LIN {X 0,Y 561.925,Z 555.197,A -85,B 0,C 180,E1 23264.855,E2 23264.855} C_VEL
LIN {X 0,Y 556.001,Z 546.029,A -85,B 0,C 180,E1 23264.105,E2 23264.105} C_VEL
LIN {X 0,Y 547.752,Z 527.565,A -85,B 0,C 180,E1 23261.432,E2 23261.432} C_VEL
LIN {X 0,Y 541.209,Z 514.277,A -85,B 0,C 180,E1 23259.278,E2 23259.278} C_VEL
LIN {X 0,Y 538.784,Z 509.459,A -85,B 0,C 180,E1 23258.452,E2 23258.452} C_VEL
LIN {X 0,Y 537.627,Z 506.4,A -85,B 0,C 180,E1 23257.909,E2 23257.909} C_VEL
LIN {X 0,Y 537.605,Z 506.203,A -85,B 0,C 180,E1 23254.522,E2 23254.522} C_VEL
LIN {X 0,Y 537.577,Z 506.243,A -85,B 0,C 180,E1 23251.137,E2 23251.137} C_VEL
LIN {X 0,Y 537.625,Z 506.246,A -85,B 0,C 180,E1 23247.828,E2 23247.828} C_VEL
LIN {X 0,Y 537.593,Z 506.246,A -85,B 0,C 180,E1 23244.505,E2 23244.505} C_VEL
LIN {X 0,Y 537.586,Z 506.245,A -85,B 0,C 180,E1 23241.037,E2 23241.037} C_VEL
LIN {X 0,Y 537.626,Z 506.247,A -85,B 0,C 180,E1 23237.759,E2 23237.759} C_VEL
LIN {X 0,Y 537.584,Z 506.265,A -85,B 0,C 180,E1 23234.432,E2 23234.432} C_VEL
LIN {X 0,Y 537.607,Z 506.257,A -85,B 0,C 180,E1 23231.044,E2 23231.044} C_VEL
LIN {X 0,Y 537.621,Z 506.234,A -85,B 0,C 180,E1 23227.696,E2 23227.696} C_VEL
LIN {X 0,Y 537.586,Z 506.247,A -85,B 0,C 180,E1 23224.374,E2 23224.374} C_VEL
LIN {X 0,Y 537.629,Z 506.263,A -85,B 0,C 180,E1 23220.959,E2 23220.959} C_VEL
LIN {X 0,Y 537.61,Z 506.254,A -85,B 0,C 180,E1 23217.548,E2 23217.548} C_VEL
LIN {X 0,Y 537.589,Z 506.241,A -85,B 0,C 180,E1 23214.128,E2 23214.128} C_VEL
LIN {X 0,Y 537.624,Z 506.249,A -85,B 0,C 180,E1 23210.796,E2 23210.796} C_VEL
LIN {X 0,Y 537.603,Z 506.263,A -85,B 0,C 180,E1 23207.431,E2 23207.431} C_VEL
LIN {X 0,Y 537.601,Z 506.253,A -85,B 0,C 180,E1 23204.022,E2 23204.022} C_VEL
LIN {X 0,Y 537.623,Z 506.24,A -85,B 0,C 180,E1 23200.667,E2 23200.667} C_VEL
LIN {X 0,Y 537.593,Z 506.245,A -85,B 0,C 180,E1 23197.356,E2 23197.356} C_VEL
LIN {X 0,Y 537.617,Z 506.248,A -85,B 0,C 180,E1 23193.933,E2 23193.933} C_VEL
LIN {X 0,Y 537.626,Z 506.251,A -85,B 0,C 180,E1 23190.501,E2 23190.501} C_VEL
LIN {X 0,Y 537.598,Z 506.252,A -85,B 0,C 180,E1 23187.105,E2 23187.105} C_VEL
LIN {X 0,Y 537.617,Z 506.22,A -85,B 0,C 180,E1 23183.741,E2 23183.741} C_VEL
LIN {X 0,Y 537.653,Z 506.458,A -85,B 0,C 180,E1 23181.617,E2 23181.617} C_VEL
LIN {X 0,Y 539.006,Z 509.849,A -85,B 0,C 180,E1 23181.009,E2 23181.009} C_VEL
LIN {X 0,Y 542.365,Z 516.8,A -85,B 0,C 180,E1 23179.815,E2 23179.815} C_VEL
LIN {X 0,Y 547.829,Z 528.287,A -85,B 0,C 180,E1 23177.945,E2 23177.945} C_VEL
LIN {X 0,Y 555.394,Z 545.389,A -85,B 0,C 180,E1 23175.402,E2 23175.402} C_VEL
LIN {X 0,Y 563.246,Z 565.031,A -85,B 0,C 180,E1 23172.772,E2 23172.772} C_VEL
LIN {X 0,Y 566.973,Z 575.356,A -85,B 0,C 180,E1 23171.498,E2 23171.498} C_VEL
LIN {X 0,Y 562.357,Z 618.194,A -85,B 0,C 180,E1 23168.165,E2 23168.165} C_VEL
LIN {X 0,Y 560.863,Z 634.529,A -85,B 0,C 180,E1 23166.942,E2 23166.942} C_VEL
LIN {X 0,Y 569.797,Z 686.668,A -85,B 0,C 180,E1 23165.398,E2 23165.398} C_VEL
LIN {X 0,Y 570.048,Z 691.209,A -85,B 0,C 180,E1 23165.312,E2 23165.312} C_VEL
LIN {X 0,Y 566.724,Z 874.265,A -85,B 0,C 180,E1 23162.984,E2 23162.984} C_VEL
LIN {X 0,Y 565.8,Z 881.967,A -85,B 0,C 180,E1 23162.947,E2 23162.947} C_VEL
LIN {X 0,Y 560.396,Z 902.487,A -85,B 0,C 180,E1 23163.067,E2 23163.067} C_VEL
LIN {X 0,Y 559.68,Z 909.097,A -85,B 0,C 180,E1 23163.029,E2 23163.029} C_VEL
LIN {X 0,Y 558.653,Z 955.968,A -85,B 0,C 180,E1 23162.406,E2 23162.406} C_VEL
LIN {X 0,Y 557.346,Z 977.728,A -85,B 0,C 180,E1 23161.949,E2 23161.949} C_VEL
LIN {X 0,Y 555.599,Z 999.514,A -85,B 0,C 180,E1 23161.308,E2 23161.308} C_VEL
LIN {X 0,Y 553.64,Z 1019.236,A -85,B 0,C 180,E1 23160.556,E2 23160.556} C_VEL
LIN {X 0,Y 551.275,Z 1038.849,A -85,B 0,C 180,E1 23159.619,E2 23159.619} C_VEL
LIN {X 0,Y 548.706,Z 1058.021,A -85,B 0,C 180,E1 23158.517,E2 23158.517} C_VEL
LIN {X 0,Y 545.967,Z 1076.282,A -85,B 0,C 180,E1 23157.248,E2 23157.248} C_VEL
LIN {X 0,Y 543.046,Z 1094.447,A -85,B 0,C 180,E1 23155.755,E2 23155.755} C_VEL
LIN {X 0,Y 540.28,Z 1111.162,A -85,B 0,C 180,E1 23154.141,E2 23154.141} C_VEL
LIN {X 0,Y 537.664,Z 1126.3,A -85,B 0,C 180,E1 23152.409,E2 23152.409} C_VEL
LIN {X 0,Y 535.194,Z 1140.977,A -85,B 0,C 180,E1 23150.448,E2 23150.448} C_VEL
LIN {X 0,Y 533.163,Z 1153.579,A -85,B 0,C 180,E1 23148.477,E2 23148.477} C_VEL
LIN {X 0,Y 531.424,Z 1164.997,A -85,B 0,C 180,E1 23146.345,E2 23146.345} C_VEL
LIN {X 0,Y 530.014,Z 1175.618,A -85,B 0,C 180,E1 23143.973,E2 23143.973} C_VEL
LIN {X 0,Y 529.079,Z 1184.103,A -85,B 0,C 180,E1 23141.666,E2 23141.666} C_VEL
LIN {X 0,Y 528.47,Z 1191.036,A -85,B 0,C 180,E1 23139.254,E2 23139.254} C_VEL
LIN {X 0,Y 528.122,Z 1196.488,A -85,B 0,C 180,E1 23136.741,E2 23136.741} C_VEL
LIN {X 0,Y 527.995,Z 1200.109,A -85,B 0,C 180,E1 23134.344,E2 23134.344} C_VEL
LIN {X 0,Y 527.948,Z 1202.071,A -85,B 0,C 180,E1 23131.954,E2 23131.954} C_VEL
LIN {X 0,Y 527.931,Z 1202.564,A -85,B 0,C 180,E1 23129.457,E2 23129.457} C_VEL
LIN {X 0,Y 527.954,Z 1201.551,A -85,B 0,C 180,E1 23127.069,E2 23127.069} C_VEL
LIN {X 0,Y 528.023,Z 1198.914,A -85,B 0,C 180,E1 23124.676,E2 23124.676} C_VEL
LIN {X 0,Y 528.229,Z 1194.547,A -85,B 0,C 180,E1 23122.167,E2 23122.167} C_VEL
LIN {X 0,Y 528.63,Z 1188.98,A -85,B 0,C 180,E1 23119.869,E2 23119.869} C_VEL
LIN {X 0,Y 529.31,Z 1181.744,A -85,B 0,C 180,E1 23117.564,E2 23117.564} C_VEL
LIN {X 0,Y 530.377,Z 1172.832,A -85,B 0,C 180,E1 23115.256,E2 23115.256} C_VEL
LIN {X 0,Y 531.807,Z 1162.469,A -85,B 0,C 180,E1 23113.057,E2 23113.057} C_VEL
LIN {X 0,Y 533.591,Z 1150.767,A -85,B 0,C 180,E1 23110.971,E2 23110.971} C_VEL
LIN {X 0,Y 535.735,Z 1137.851,A -85,B 0,C 180,E1 23109.002,E2 23109.002} C_VEL
LIN {X 0,Y 538.171,Z 1123.45,A -85,B 0,C 180,E1 23107.151,E2 23107.151} C_VEL
LIN {X 0,Y 540.926,Z 1107.216,A -85,B 0,C 180,E1 23105.366,E2 23105.366} C_VEL
LIN {X 0,Y 543.725,Z 1090.665,A -85,B 0,C 180,E1 23103.811,E2 23103.811} C_VEL
LIN {X 0,Y 546.464,Z 1073.135,A -85,B 0,C 180,E1 23102.425,E2 23102.425} C_VEL
LIN {X 0,Y 549.38,Z 1053.232,A -85,B 0,C 180,E1 23101.097,E2 23101.097} C_VEL
LIN {X 0,Y 552.014,Z 1033.48,A -85,B 0,C 180,E1 23100.006,E2 23100.006} C_VEL
LIN {X 0,Y 554.239,Z 1013.599,A -85,B 0,C 180,E1 23099.12,E2 23099.12} C_VEL
LIN {X 0,Y 556.28,Z 991.947,A -85,B 0,C 180,E1 23098.351,E2 23098.351} C_VEL
LIN {X 0,Y 557.841,Z 971.023,A -85,B 0,C 180,E1 23097.796,E2 23097.796} C_VEL
LIN {X 0,Y 558.926,Z 948.814,A -85,B 0,C 180,E1 23097.393,E2 23097.393} C_VEL
LIN {X 0,Y 563.835,Z 689.521,A -85,B 0,C 180,E1 23094.052,E2 23094.052} C_VEL
LIN {X 0,Y 555.184,Z 638.455,A -85,B 0,C 180,E1 23092.521,E2 23092.521} C_VEL
LIN {X 0,Y 554.334,Z 632.446,A -85,B 0,C 180,E1 23092.305,E2 23092.305} C_VEL
LIN {X 0,Y 559.067,Z 589.044,A -85,B 0,C 180,E1 23088.91,E2 23088.91} C_VEL
LIN {X 0,Y 560.277,Z 578.706,A -85,B 0,C 180,E1 23088.09,E2 23088.09} C_VEL
LIN {X 0,Y 552.971,Z 559.337,A -85,B 0,C 180,E1 23085.582,E2 23085.582} C_VEL
LIN {X 0,Y 545.415,Z 541.259,A -85,B 0,C 180,E1 23082.992,E2 23082.992} C_VEL
LIN {X 0,Y 538.993,Z 527.2,A -85,B 0,C 180,E1 23080.768,E2 23080.768} C_VEL
LIN {X 0,Y 533.777,Z 515.999,A -85,B 0,C 180,E1 23078.869,E2 23078.869} C_VEL
LIN {X 0,Y 530.962,Z 510.631,A -85,B 0,C 180,E1 23077.873,E2 23077.873} C_VEL
LIN {X 0,Y 529.693,Z 507.425,A -85,B 0,C 180,E1 23077.26,E2 23077.26} C_VEL
LIN {X 0,Y 529.686,Z 507.237,A -85,B 0,C 180,E1 23073.97,E2 23073.97} C_VEL
LIN {X 0,Y 529.655,Z 507.239,A -85,B 0,C 180,E1 23070.592,E2 23070.592} C_VEL
LIN {X 0,Y 529.676,Z 507.234,A -85,B 0,C 180,E1 23067.183,E2 23067.183} C_VEL
LIN {X 0,Y 529.685,Z 507.233,A -85,B 0,C 180,E1 23063.722,E2 23063.722} C_VEL
LIN {X 0,Y 529.652,Z 507.252,A -85,B 0,C 180,E1 23060.441,E2 23060.441} C_VEL
LIN {X 0,Y 529.683,Z 507.25,A -85,B 0,C 180,E1 23057.014,E2 23057.014} C_VEL
LIN {X 0,Y 529.681,Z 507.239,A -85,B 0,C 180,E1 23053.537,E2 23053.537} C_VEL
LIN {X 0,Y 529.647,Z 507.228,A -85,B 0,C 180,E1 23050.112,E2 23050.112} C_VEL
LIN {X 0,Y 529.683,Z 507.234,A -85,B 0,C 180,E1 23046.721,E2 23046.721} C_VEL
LIN {X 0,Y 529.677,Z 507.253,A -85,B 0,C 180,E1 23043.247,E2 23043.247} C_VEL
LIN {X 0,Y 529.646,Z 507.246,A -85,B 0,C 180,E1 23039.892,E2 23039.892} C_VEL
LIN {X 0,Y 529.681,Z 507.225,A -85,B 0,C 180,E1 23036.537,E2 23036.537} C_VEL
LIN {X 0,Y 529.659,Z 507.242,A -85,B 0,C 180,E1 23033.17,E2 23033.17} C_VEL
LIN {X 0,Y 529.647,Z 507.254,A -85,B 0,C 180,E1 23029.668,E2 23029.668} C_VEL
LIN {X 0,Y 529.69,Z 507.238,A -85,B 0,C 180,E1 23026.24,E2 23026.24} C_VEL
LIN {X 0,Y 529.647,Z 507.231,A -85,B 0,C 180,E1 23022.985,E2 23022.985} C_VEL
LIN {X 0,Y 529.65,Z 507.235,A -85,B 0,C 180,E1 23019.559,E2 23019.559} C_VEL
LIN {X 0,Y 529.687,Z 507.239,A -85,B 0,C 180,E1 23016.277,E2 23016.277} C_VEL
LIN {X 0,Y 529.642,Z 507.255,A -85,B 0,C 180,E1 23012.937,E2 23012.937} C_VEL
LIN {X 0,Y 529.68,Z 507.251,A -85,B 0,C 180,E1 23009.608,E2 23009.608} C_VEL
LIN {X 0,Y 529.652,Z 507.179,A -85,B 0,C 180,E1 23006.288,E2 23006.288} C_VEL
LIN {X 0,Y 529.68,Z 507.481,A -85,B 0,C 180,E1 23003.086,E2 23003.086} C_VEL
LIN {X 0,Y 531.21,Z 511.069,A -85,B 0,C 180,E1 23002.42,E2 23002.42} C_VEL
LIN {X 0,Y 534.623,Z 517.979,A -85,B 0,C 180,E1 23001.204,E2 23001.204} C_VEL
LIN {X 0,Y 540.143,Z 529.123,A -85,B 0,C 180,E1 22999.337,E2 22999.337} C_VEL
LIN {X 0,Y 548.485,Z 547.475,A -85,B 0,C 180,E1 22996.576,E2 22996.576} C_VEL
LIN {X 0,Y 563.622,Z 570.87,A -85,B 0,C 180,E1 22994.724,E2 22994.724} C_VEL
LIN {X 0,Y 570.245,Z 582.252,A -85,B 0,C 180,E1 22993.946,E2 22993.946} C_VEL
LIN {X 0,Y 562.926,Z 822.165,A -85,B 0,C 180,E1 22990.433,E2 22990.433} C_VEL
LIN {X 0,Y 559.893,Z 922.618,A -85,B 0,C 180,E1 22988.935,E2 22988.935} C_VEL
LIN {X 0,Y 558.457,Z 947.453,A -85,B 0,C 180,E1 22988.394,E2 22988.394} C_VEL
LIN {X 0,Y 556.833,Z 969.384,A -85,B 0,C 180,E1 22987.761,E2 22987.761} C_VEL
LIN {X 0,Y 554.701,Z 993.174,A -85,B 0,C 180,E1 22986.887,E2 22986.887} C_VEL
LIN {X 0,Y 552.675,Z 1012.791,A -85,B 0,C 180,E1 22986.013,E2 22986.013} C_VEL
LIN {X 0,Y 550.066,Z 1035.704,A -85,B 0,C 180,E1 22984.803,E2 22984.803} C_VEL
LIN {X 0,Y 547.495,Z 1056.007,A -85,B 0,C 180,E1 22983.534,E2 22983.534} C_VEL
LIN {X 0,Y 544.725,Z 1077.173,A -85,B 0,C 180,E1 22982,E2 22982} C_VEL
LIN {X 0,Y 542.149,Z 1095.835,A -85,B 0,C 180,E1 22980.43,E2 22980.43} C_VEL
LIN {X 0,Y 539.441,Z 1115.215,A -85,B 0,C 180,E1 22978.568,E2 22978.568} C_VEL
LIN {X 0,Y 537.189,Z 1131.451,A -85,B 0,C 180,E1 22976.771,E2 22976.771} C_VEL
LIN {X 0,Y 534.918,Z 1148.46,A -85,B 0,C 180,E1 22974.634,E2 22974.634} C_VEL
LIN {X 0,Y 533.128,Z 1162.417,A -85,B 0,C 180,E1 22972.611,E2 22972.611} C_VEL
LIN {X 0,Y 531.533,Z 1176.087,A -85,B 0,C 180,E1 22970.365,E2 22970.365} C_VEL
LIN {X 0,Y 530.254,Z 1188.25,A -85,B 0,C 180,E1 22968.013,E2 22968.013} C_VEL
LIN {X 0,Y 529.33,Z 1198.776,A -85,B 0,C 180,E1 22965.671,E2 22965.671} C_VEL
LIN {X 0,Y 528.67,Z 1207.8,A -85,B 0,C 180,E1 22963.229,E2 22963.229} C_VEL
LIN {X 0,Y 528.281,Z 1214.596,A -85,B 0,C 180,E1 22961.02,E2 22961.02} C_VEL
LIN {X 0,Y 528.051,Z 1220.963,A -85,B 0,C 180,E1 22958.383,E2 22958.383} C_VEL
LIN {X 0,Y 527.958,Z 1224.858,A -85,B 0,C 180,E1 22956.197,E2 22956.197} C_VEL
LIN {X 0,Y 527.92,Z 1227.839,A -85,B 0,C 180,E1 22953.801,E2 22953.801} C_VEL
LIN {X 0,Y 527.915,Z 1229.386,A -85,B 0,C 180,E1 22951.194,E2 22951.194} C_VEL
LIN {X 0,Y 527.906,Z 1229.435,A -85,B 0,C 180,E1 22949.023,E2 22949.023} C_VEL
LIN {X 0,Y 527.911,Z 1228.229,A -85,B 0,C 180,E1 22946.634,E2 22946.634} C_VEL
LIN {X 0,Y 527.95,Z 1225.204,A -85,B 0,C 180,E1 22944.021,E2 22944.021} C_VEL
LIN {X 0,Y 528.023,Z 1221.407,A -85,B 0,C 180,E1 22941.835,E2 22941.835} C_VEL
LIN {X 0,Y 528.257,Z 1215.237,A -85,B 0,C 180,E1 22939.2,E2 22939.2} C_VEL
LIN {X 0,Y 528.645,Z 1208.18,A -85,B 0,C 180,E1 22936.882,E2 22936.882} C_VEL
LIN {X 0,Y 529.293,Z 1199.229,A -85,B 0,C 180,E1 22934.44,E2 22934.44} C_VEL
LIN {X 0,Y 530.202,Z 1188.797,A -85,B 0,C 180,E1 22932.098,E2 22932.098} C_VEL
LIN {X 0,Y 531.393,Z 1177.294,A -85,B 0,C 180,E1 22929.859,E2 22929.859} C_VEL
LIN {X 0,Y 533.042,Z 1163.148,A -85,B 0,C 180,E1 22927.502,E2 22927.502} C_VEL
LIN {X 0,Y 534.803,Z 1149.258,A -85,B 0,C 180,E1 22925.478,E2 22925.478} C_VEL
LIN {X 0,Y 537.069,Z 1132.352,A -85,B 0,C 180,E1 22923.335,E2 22923.335} C_VEL
LIN {X 0,Y 539.358,Z 1115.746,A -85,B 0,C 180,E1 22921.49,E2 22921.49} C_VEL
LIN {X 0,Y 542.037,Z 1096.607,A -85,B 0,C 180,E1 22919.64,E2 22919.64} C_VEL
LIN {X 0,Y 544.449,Z 1079.056,A -85,B 0,C 180,E1 22918.154,E2 22918.154} C_VEL
LIN {X 0,Y 547.386,Z 1056.795,A -85,B 0,C 180,E1 22916.521,E2 22916.521} C_VEL
LIN {X 0,Y 549.937,Z 1036.58,A -85,B 0,C 180,E1 22915.251,E2 22915.251} C_VEL
LIN {X 0,Y 552.549,Z 1013.879,A -85,B 0,C 180,E1 22914.042,E2 22914.042} C_VEL
LIN {X 0,Y 554.561,Z 994.395,A -85,B 0,C 180,E1 22913.167,E2 22913.167} C_VEL
LIN {X 0,Y 556.735,Z 970.49,A -85,B 0,C 180,E1 22912.277,E2 22912.277} C_VEL
LIN {X 0,Y 558.383,Z 948.318,A -85,B 0,C 180,E1 22911.632,E2 22911.632} C_VEL
LIN {X 0,Y 559.814,Z 924.247,A -85,B 0,C 180,E1 22911.096,E2 22911.096} C_VEL
LIN {X 0,Y 561.907,Z 856.989,A -85,B 0,C 180,E1 22910.083,E2 22910.083} C_VEL
LIN {X 0,Y 569.311,Z 611.877,A -85,B 0,C 180,E1 22906.486,E2 22906.486} C_VEL
LIN {X 0,Y 570.092,Z 581.629,A -85,B 0,C 180,E1 22906.035,E2 22906.035} C_VEL
LIN {X 0,Y 555.994,Z 558.916,A -85,B 0,C 180,E1 22904.375,E2 22904.375} C_VEL
LIN {X 0,Y 548.434,Z 547.379,A -85,B 0,C 180,E1 22903.42,E2 22903.42} C_VEL
LIN {X 0,Y 541.343,Z 531.833,A -85,B 0,C 180,E1 22901.099,E2 22901.099} C_VEL
LIN {X 0,Y 535.554,Z 519.76,A -85,B 0,C 180,E1 22899.128,E2 22899.128} C_VEL
LIN {X 0,Y 531.524,Z 511.479,A -85,B 0,C 180,E1 22897.69,E2 22897.69} C_VEL
LIN {X 0,Y 529.747,Z 507.875,A -85,B 0,C 180,E1 22897.021,E2 22897.021} C_VEL
LIN {X 0,Y 529.663,Z 507.28,A -85,B 0,C 180,E1 22896.758,E2 22896.758} C_VEL
LIN {X 0,Y 529.634,Z 507.18,A -85,B 0,C 180,E1 22893.324,E2 22893.324} C_VEL
LIN {X 0,Y 529.694,Z 507.251,A -85,B 0,C 180,E1 22889.956,E2 22889.956} C_VEL
LIN {X 0,Y 529.649,Z 507.256,A -85,B 0,C 180,E1 22886.699,E2 22886.699} C_VEL
LIN {X 0,Y 529.651,Z 507.257,A -85,B 0,C 180,E1 22883.17,E2 22883.17} C_VEL
LIN {X 0,Y 529.688,Z 507.24,A -85,B 0,C 180,E1 22879.864,E2 22879.864} C_VEL
LIN {X 0,Y 529.646,Z 507.234,A -85,B 0,C 180,E1 22876.45,E2 22876.45} C_VEL
LIN {X 0,Y 529.657,Z 507.23,A -85,B 0,C 180,E1 22872.982,E2 22872.982} C_VEL
LIN {X 0,Y 529.686,Z 507.243,A -85,B 0,C 180,E1 22869.562,E2 22869.562} C_VEL
LIN {X 0,Y 529.65,Z 507.252,A -85,B 0,C 180,E1 22866.177,E2 22866.177} C_VEL
LIN {X 0,Y 529.663,Z 507.232,A -85,B 0,C 180,E1 22862.705,E2 22862.705} C_VEL
LIN {X 0,Y 529.688,Z 507.228,A -85,B 0,C 180,E1 22859.351,E2 22859.351} C_VEL
LIN {X 0,Y 529.65,Z 507.251,A -85,B 0,C 180,E1 22855.995,E2 22855.995} C_VEL
LIN {X 0,Y 529.678,Z 507.246,A -85,B 0,C 180,E1 22852.516,E2 22852.516} C_VEL
LIN {X 0,Y 529.681,Z 507.226,A -85,B 0,C 180,E1 22849.119,E2 22849.119} C_VEL
LIN {X 0,Y 529.65,Z 507.233,A -85,B 0,C 180,E1 22845.793,E2 22845.793} C_VEL
LIN {X 0,Y 529.686,Z 507.245,A -85,B 0,C 180,E1 22842.413,E2 22842.413} C_VEL
LIN {X 0,Y 529.682,Z 507.251,A -85,B 0,C 180,E1 22838.982,E2 22838.982} C_VEL
LIN {X 0,Y 529.658,Z 507.25,A -85,B 0,C 180,E1 22835.579,E2 22835.579} C_VEL
LIN {X 0,Y 529.685,Z 507.241,A -85,B 0,C 180,E1 22832.208,E2 22832.208} C_VEL
LIN {X 0,Y 529.681,Z 507.245,A -85,B 0,C 180,E1 22828.726,E2 22828.726} C_VEL
LIN {X 0,Y 529.661,Z 507.253,A -85,B 0,C 180,E1 22825.242,E2 22825.242} C_VEL
LIN {X 0,Y 529.707,Z 507.46,A -85,B 0,C 180,E1 22822.605,E2 22822.605} C_VEL
LIN {X 0,Y 531.368,Z 511.221,A -85,B 0,C 180,E1 22821.887,E2 22821.887} C_VEL
LIN {X 0,Y 538.141,Z 525.268,A -85,B 0,C 180,E1 22819.434,E2 22819.434} C_VEL
LIN {X 0,Y 545.188,Z 540.732,A -85,B 0,C 180,E1 22816.979,E2 22816.979} C_VEL
LIN {X 0,Y 552.728,Z 558.775,A -85,B 0,C 180,E1 22814.393,E2 22814.393} C_VEL
LIN {X 0,Y 560.044,Z 578.118,A -85,B 0,C 180,E1 22811.883,E2 22811.883} C_VEL
LIN {X 0,Y 560.052,Z 580.316,A -85,B 0,C 180,E1 22811.684,E2 22811.684} C_VEL
LIN {X 0,Y 555.207,Z 623.665,A -85,B 0,C 180,E1 22808.28,E2 22808.28} C_VEL
LIN {X 0,Y 554.32,Z 633.589,A -85,B 0,C 180,E1 22807.537,E2 22807.537} C_VEL
LIN {X 0,Y 563.364,Z 686.902,A -85,B 0,C 180,E1 22805.925,E2 22805.925} C_VEL
LIN {X 0,Y 563.818,Z 691.587,A -85,B 0,C 180,E1 22805.818,E2 22805.818} C_VEL
LIN {X 0,Y 559.68,Z 909.097,A -85,B 0,C 180,E1 22803.029,E2 22803.029} C_VEL
LIN {X 0,Y 558.767,Z 916.801,A -85,B 0,C 180,E1 22802.993,E2 22802.993} C_VEL
LIN {X 0,Y 553.38,Z 937.323,A -85,B 0,C 180,E1 22803.119,E2 22803.119} C_VEL
LIN {X 0,Y 552.584,Z 943.921,A -85,B 0,C 180,E1 22803.072,E2 22803.072} C_VEL
LIN {X 0,Y 551.636,Z 965.523,A -85,B 0,C 180,E1 22802.708,E2 22802.708} C_VEL
LIN {X 0,Y 550.035,Z 987.611,A -85,B 0,C 180,E1 22802.159,E2 22802.159} C_VEL
LIN {X 0,Y 548.151,Z 1008.166,A -85,B 0,C 180,E1 22801.476,E2 22801.476} C_VEL
LIN {X 0,Y 545.831,Z 1028.216,A -85,B 0,C 180,E1 22800.613,E2 22800.613} C_VEL
LIN {X 0,Y 543.086,Z 1049.13,A -85,B 0,C 180,E1 22799.504,E2 22799.504} C_VEL
LIN {X 0,Y 540.369,Z 1067.436,A -85,B 0,C 180,E1 22798.334,E2 22798.334} C_VEL
LIN {X 0,Y 537.403,Z 1085.622,A -85,B 0,C 180,E1 22796.939,E2 22796.939} C_VEL
LIN {X 0,Y 534.387,Z 1103.264,A -85,B 0,C 180,E1 22795.345,E2 22795.345} C_VEL
LIN {X 0,Y 531.538,Z 1119.32,A -85,B 0,C 180,E1 22793.636,E2 22793.636} C_VEL
LIN {X 0,Y 528.992,Z 1133.489,A -85,B 0,C 180,E1 22791.861,E2 22791.861} C_VEL
LIN {X 0,Y 526.611,Z 1147.186,A -85,B 0,C 180,E1 22789.868,E2 22789.868} C_VEL
LIN {X 0,Y 524.572,Z 1159.409,A -85,B 0,C 180,E1 22787.756,E2 22787.756} C_VEL
LIN {X 0,Y 522.887,Z 1170.516,A -85,B 0,C 180,E1 22785.468,E2 22785.468} C_VEL
LIN {X 0,Y 521.673,Z 1179.798,A -85,B 0,C 180,E1 22783.173,E2 22783.173} C_VEL
LIN {X 0,Y 520.848,Z 1187.373,A -85,B 0,C 180,E1 22780.844,E2 22780.844} C_VEL
LIN {X 0,Y 520.336,Z 1193.613,A -85,B 0,C 180,E1 22778.397,E2 22778.397} C_VEL
LIN {X 0,Y 520.068,Z 1198.251,A -85,B 0,C 180,E1 22775.959,E2 22775.959} C_VEL
LIN {X 0,Y 519.969,Z 1201.174,A -85,B 0,C 180,E1 22773.528,E2 22773.528} C_VEL
LIN {X 0,Y 519.943,Z 1202.665,A -85,B 0,C 180,E1 22770.992,E2 22770.992} C_VEL
LIN {X 0,Y 519.938,Z 1202.62,A -85,B 0,C 180,E1 22768.678,E2 22768.678} C_VEL
LIN {X 0,Y 519.972,Z 1201.051,A -85,B 0,C 180,E1 22766.251,E2 22766.251} C_VEL
LIN {X 0,Y 520.082,Z 1198.044,A -85,B 0,C 180,E1 22763.82,E2 22763.82} C_VEL
LIN {X 0,Y 520.362,Z 1193.333,A -85,B 0,C 180,E1 22761.38,E2 22761.38} C_VEL
LIN {X 0,Y 520.924,Z 1186.646,A -85,B 0,C 180,E1 22758.822,E2 22758.822} C_VEL
LIN {X 0,Y 521.794,Z 1178.875,A -85,B 0,C 180,E1 22756.481,E2 22756.481} C_VEL
LIN {X 0,Y 523.09,Z 1169.182,A -85,B 0,C 180,E1 22754.137,E2 22754.137} C_VEL
LIN {X 0,Y 524.785,Z 1158.077,A -85,B 0,C 180,E1 22751.907,E2 22751.907} C_VEL
LIN {X 0,Y 526.881,Z 1145.646,A -85,B 0,C 180,E1 22749.795,E2 22749.795} C_VEL
LIN {X 0,Y 529.176,Z 1132.518,A -85,B 0,C 180,E1 22747.914,E2 22747.914} C_VEL
LIN {X 0,Y 531.991,Z 1116.786,A -85,B 0,C 180,E1 22745.987,E2 22745.987} C_VEL
LIN {X 0,Y 534.893,Z 1100.574,A -85,B 0,C 180,E1 22744.293,E2 22744.293} C_VEL
LIN {X 0,Y 537.796,Z 1083.411,A -85,B 0,C 180,E1 22742.783,E2 22742.783} C_VEL
LIN {X 0,Y 540.915,Z 1063.933,A -85,B 0,C 180,E1 22741.336,E2 22741.336} C_VEL
LIN {X 0,Y 543.687,Z 1045.202,A -85,B 0,C 180,E1 22740.168,E2 22740.168} C_VEL
LIN {X 0,Y 546.228,Z 1025.211,A -85,B 0,C 180,E1 22739.152,E2 22739.152} C_VEL
LIN {X 0,Y 548.611,Z 1003.695,A -85,B 0,C 180,E1 22738.271,E2 22738.271} C_VEL
LIN {X 0,Y 550.433,Z 983.394,A -85,B 0,C 180,E1 22737.622,E2 22737.622} C_VEL
LIN {X 0,Y 551.866,Z 961.836,A -85,B 0,C 180,E1 22737.126,E2 22737.126} C_VEL
LIN {X 0,Y 552.758,Z 937.791,A -85,B 0,C 180,E1 22736.751,E2 22736.751} C_VEL
LIN {X 0,Y 557.622,Z 690.877,A -85,B 0,C 180,E1 22733.546,E2 22733.546} C_VEL
LIN {X 0,Y 548.873,Z 638.521,A -85,B 0,C 180,E1 22731.947,E2 22731.947} C_VEL
LIN {X 0,Y 547.829,Z 631.704,A -85,B 0,C 180,E1 22731.705,E2 22731.705} C_VEL
LIN {X 0,Y 552.896,Z 587.57,A -85,B 0,C 180,E1 22728.211,E2 22728.211} C_VEL
LIN {X 0,Y 553.563,Z 582.2,A -85,B 0,C 180,E1 22727.781,E2 22727.781} C_VEL
LIN {X 0,Y 546.327,Z 562.98,A -85,B 0,C 180,E1 22725.245,E2 22725.245} C_VEL
LIN {X 0,Y 538.896,Z 545.02,A -85,B 0,C 180,E1 22722.628,E2 22722.628} C_VEL
LIN {X 0,Y 531.608,Z 529.059,A -85,B 0,C 180,E1 22720.036,E2 22720.036} C_VEL
LIN {X 0,Y 525.868,Z 516.941,A -85,B 0,C 180,E1 22717.891,E2 22717.891} C_VEL
LIN {X 0,Y 523.101,Z 511.787,A -85,B 0,C 180,E1 22716.885,E2 22716.885} C_VEL
LIN {X 0,Y 521.77,Z 508.433,A -85,B 0,C 180,E1 22716.22,E2 22716.22} C_VEL
LIN {X 0,Y 521.716,Z 508.229,A -85,B 0,C 180,E1 22712.846,E2 22712.846} C_VEL
LIN {X 0,Y 521.749,Z 508.226,A -85,B 0,C 180,E1 22709.507,E2 22709.507} C_VEL
LIN {X 0,Y 521.734,Z 508.224,A -85,B 0,C 180,E1 22706.032,E2 22706.032} C_VEL
LIN {X 0,Y 521.712,Z 508.221,A -85,B 0,C 180,E1 22702.539,E2 22702.539} C_VEL
LIN {X 0,Y 521.744,Z 508.215,A -85,B 0,C 180,E1 22699.13,E2 22699.13} C_VEL
LIN {X 0,Y 521.737,Z 508.222,A -85,B 0,C 180,E1 22695.678,E2 22695.678} C_VEL
LIN {X 0,Y 521.712,Z 508.244,A -85,B 0,C 180,E1 22692.202,E2 22692.202} C_VEL
LIN {X 0,Y 521.742,Z 508.238,A -85,B 0,C 180,E1 22688.708,E2 22688.708} C_VEL
LIN {X 0,Y 521.738,Z 508.217,A -85,B 0,C 180,E1 22685.278,E2 22685.278} C_VEL
LIN {X 0,Y 521.704,Z 508.224,A -85,B 0,C 180,E1 22681.867,E2 22681.867} C_VEL
LIN {X 0,Y 521.741,Z 508.238,A -85,B 0,C 180,E1 22678.463,E2 22678.463} C_VEL
LIN {X 0,Y 521.732,Z 508.231,A -85,B 0,C 180,E1 22675.053,E2 22675.053} C_VEL
LIN {X 0,Y 521.703,Z 508.216,A -85,B 0,C 180,E1 22671.735,E2 22671.735} C_VEL
LIN {X 0,Y 521.745,Z 508.222,A -85,B 0,C 180,E1 22668.312,E2 22668.312} C_VEL
LIN {X 0,Y 521.721,Z 508.242,A -85,B 0,C 180,E1 22664.891,E2 22664.891} C_VEL
LIN {X 0,Y 521.707,Z 508.241,A -85,B 0,C 180,E1 22661.449,E2 22661.449} C_VEL
LIN {X 0,Y 521.755,Z 508.224,A -85,B 0,C 180,E1 22658.049,E2 22658.049} C_VEL
LIN {X 0,Y 521.711,Z 508.223,A -85,B 0,C 180,E1 22654.698,E2 22654.698} C_VEL
LIN {X 0,Y 521.703,Z 508.226,A -85,B 0,C 180,E1 22651.245,E2 22651.245} C_VEL
LIN {X 0,Y 521.74,Z 508.18,A -85,B 0,C 180,E1 22648.066,E2 22648.066} C_VEL
LIN {X 0,Y 521.694,Z 508.203,A -85,B 0,C 180,E1 22644.731,E2 22644.731} C_VEL
LIN {X 0,Y 521.793,Z 508.627,A -85,B 0,C 180,E1 22644.083,E2 22644.083} C_VEL
LIN {X 0,Y 523.368,Z 512.18,A -85,B 0,C 180,E1 22643.411,E2 22643.411} C_VEL
LIN {X 0,Y 528.508,Z 522.258,A -85,B 0,C 180,E1 22641.557,E2 22641.557} C_VEL
LIN {X 0,Y 534.627,Z 535.149,A -85,B 0,C 180,E1 22639.394,E2 22639.394} C_VEL
LIN {X 0,Y 541.014,Z 548.948,A -85,B 0,C 180,E1 22637.29,E2 22637.29} C_VEL
LIN {X 0,Y 555.291,Z 570.751,A -85,B 0,C 180,E1 22635.486,E2 22635.486} C_VEL
LIN {X 0,Y 564.079,Z 585.32,A -85,B 0,C 180,E1 22634.43,E2 22634.43} C_VEL
LIN {X 0,Y 556.491,Z 824.096,A -85,B 0,C 180,E1 22630.902,E2 22630.902} C_VEL
LIN {X 0,Y 553.383,Z 922.805,A -85,B 0,C 180,E1 22629.414,E2 22629.414} C_VEL
LIN {X 0,Y 551.888,Z 947.733,A -85,B 0,C 180,E1 22628.866,E2 22628.866} C_VEL
LIN {X 0,Y 550.191,Z 969.793,A -85,B 0,C 180,E1 22628.223,E2 22628.223} C_VEL
LIN {X 0,Y 547.95,Z 993.744,A -85,B 0,C 180,E1 22627.331,E2 22627.331} C_VEL
LIN {X 0,Y 545.762,Z 1014.07,A -85,B 0,C 180,E1 22626.411,E2 22626.411} C_VEL
LIN {X 0,Y 542.945,Z 1037.449,A -85,B 0,C 180,E1 22625.147,E2 22625.147} C_VEL
LIN {X 0,Y 540.336,Z 1057.222,A -85,B 0,C 180,E1 22623.888,E2 22623.888} C_VEL
LIN {X 0,Y 537.239,Z 1079.573,A -85,B 0,C 180,E1 22622.222,E2 22622.222} C_VEL
LIN {X 0,Y 534.687,Z 1097.284,A -85,B 0,C 180,E1 22620.697,E2 22620.697} C_VEL
LIN {X 0,Y 531.806,Z 1116.785,A -85,B 0,C 180,E1 22618.771,E2 22618.771} C_VEL
LIN {X 0,Y 529.481,Z 1132.865,A -85,B 0,C 180,E1 22616.95,E2 22616.95} C_VEL
LIN {X 0,Y 526.984,Z 1150.527,A -85,B 0,C 180,E1 22614.653,E2 22614.653} C_VEL
LIN {X 0,Y 525.138,Z 1164.519,A -85,B 0,C 180,E1 22612.561,E2 22612.561} C_VEL
LIN {X 0,Y 523.4,Z 1178.669,A -85,B 0,C 180,E1 22610.112,E2 22610.112} C_VEL
LIN {X 0,Y 522.239,Z 1189.451,A -85,B 0,C 180,E1 22607.953,E2 22607.953} C_VEL
LIN {X 0,Y 521.224,Z 1200.526,A -85,B 0,C 180,E1 22605.35,E2 22605.35} C_VEL
LIN {X 0,Y 520.639,Z 1208.526,A -85,B 0,C 180,E1 22603.098,E2 22603.098} C_VEL
LIN {X 0,Y 520.212,Z 1216.079,A -85,B 0,C 180,E1 22600.521,E2 22600.521} C_VEL
LIN {X 0,Y 520.024,Z 1221.33,A -85,B 0,C 180,E1 22598.18,E2 22598.18} C_VEL
LIN {X 0,Y 519.95,Z 1225.114,A -85,B 0,C 180,E1 22595.96,E2 22595.96} C_VEL
LIN {X 0,Y 519.911,Z 1228.083,A -85,B 0,C 180,E1 22593.307,E2 22593.307} C_VEL
LIN {X 0,Y 519.909,Z 1229.227,A -85,B 0,C 180,E1 22590.992,E2 22590.992} C_VEL
LIN {X 0,Y 519.914,Z 1229.205,A -85,B 0,C 180,E1 22588.898,E2 22588.898} C_VEL
LIN {X 0,Y 519.919,Z 1227.851,A -85,B 0,C 180,E1 22586.361,E2 22586.361} C_VEL
LIN {X 0,Y 519.959,Z 1224.788,A -85,B 0,C 180,E1 22583.818,E2 22583.818} C_VEL
LIN {X 0,Y 520.062,Z 1220.688,A -85,B 0,C 180,E1 22581.487,E2 22581.487} C_VEL
LIN {X 0,Y 520.3,Z 1214.251,A -85,B 0,C 180,E1 22578.808,E2 22578.808} C_VEL
LIN {X 0,Y 520.716,Z 1207.414,A -85,B 0,C 180,E1 22576.565,E2 22576.565} C_VEL
LIN {X 0,Y 521.457,Z 1197.874,A -85,B 0,C 180,E1 22573.972,E2 22573.972} C_VEL
LIN {X 0,Y 522.418,Z 1187.729,A -85,B 0,C 180,E1 22571.683,E2 22571.683} C_VEL
LIN {X 0,Y 523.79,Z 1175.508,A -85,B 0,C 180,E1 22569.292,E2 22569.292} C_VEL
LIN {X 0,Y 525.448,Z 1161.963,A -85,B 0,C 180,E1 22567.04,E2 22567.04} C_VEL
LIN {X 0,Y 527.478,Z 1147.185,A -85,B 0,C 180,E1 22564.875,E2 22564.875} C_VEL
LIN {X 0,Y 529.74,Z 1130.927,A -85,B 0,C 180,E1 22562.822,E2 22562.822} C_VEL
LIN {X 0,Y 532.364,Z 1113.265,A -85,B 0,C 180,E1 22560.853,E2 22560.853} C_VEL
LIN {X 0,Y 535.049,Z 1094.654,A -85,B 0,C 180,E1 22559.068,E2 22559.068} C_VEL
LIN {X 0,Y 537.945,Z 1074.675,A -85,B 0,C 180,E1 22557.384,E2 22557.384} C_VEL
LIN {X 0,Y 540.711,Z 1054.365,A -85,B 0,C 180,E1 22555.924,E2 22555.924} C_VEL
LIN {X 0,Y 543.576,Z 1032.734,A -85,B 0,C 180,E1 22554.576,E2 22554.576} C_VEL
LIN {X 0,Y 546.082,Z 1010.969,A -85,B 0,C 180,E1 22553.442,E2 22553.442} C_VEL
LIN {X 0,Y 548.527,Z 987.955,A -85,B 0,C 180,E1 22552.43,E2 22552.43} C_VEL
LIN {X 0,Y 550.579,Z 964.321,A -85,B 0,C 180,E1 22551.605,E2 22551.605} C_VEL
LIN {X 0,Y 552.416,Z 939.78,A -85,B 0,C 180,E1 22550.938,E2 22550.938} C_VEL
LIN {X 0,Y 553.635,Z 916.349,A -85,B 0,C 180,E1 22550.482,E2 22550.482} C_VEL
LIN {X 0,Y 561.264,Z 671.541,A -85,B 0,C 180,E1 22546.837,E2 22546.837} C_VEL
LIN {X 0,Y 563.914,Z 584.941,A -85,B 0,C 180,E1 22545.554,E2 22545.554} C_VEL
LIN {X 0,Y 550.586,Z 563.375,A -85,B 0,C 180,E1 22543.944,E2 22543.944} C_VEL
LIN {X 0,Y 540.712,Z 548.451,A -85,B 0,C 180,E1 22542.667,E2 22542.667} C_VEL
LIN {X 0,Y 533.759,Z 533.303,A -85,B 0,C 180,E1 22540.323,E2 22540.323} C_VEL
LIN {X 0,Y 527.608,Z 520.565,A -85,B 0,C 180,E1 22538.157,E2 22538.157} C_VEL
LIN {X 0,Y 525.412,Z 516.323,A -85,B 0,C 180,E1 22537.379,E2 22537.379} C_VEL
LIN {X 0,Y 523.309,Z 512.092,A -85,B 0,C 180,E1 22536.594,E2 22536.594} C_VEL
LIN {X 0,Y 521.75,Z 508.381,A -85,B 0,C 180,E1 22535.867,E2 22535.867} C_VEL
LIN {X 0,Y 521.717,Z 508.169,A -85,B 0,C 180,E1 22532.585,E2 22532.585} C_VEL
LIN {X 0,Y 521.705,Z 508.232,A -85,B 0,C 180,E1 22529.257,E2 22529.257} C_VEL
LIN {X 0,Y 521.748,Z 508.229,A -85,B 0,C 180,E1 22525.909,E2 22525.909} C_VEL
LIN {X 0,Y 521.712,Z 508.243,A -85,B 0,C 180,E1 22522.52,E2 22522.52} C_VEL
LIN {X 0,Y 521.712,Z 508.245,A -85,B 0,C 180,E1 22519.015,E2 22519.015} C_VEL
LIN {X 0,Y 521.753,Z 508.229,A -85,B 0,C 180,E1 22515.563,E2 22515.563} C_VEL
LIN {X 0,Y 521.714,Z 508.219,A -85,B 0,C 180,E1 22512.17,E2 22512.17} C_VEL
LIN {X 0,Y 521.71,Z 508.217,A -85,B 0,C 180,E1 22508.709,E2 22508.709} C_VEL
LIN {X 0,Y 521.75,Z 508.238,A -85,B 0,C 180,E1 22505.388,E2 22505.388} C_VEL
LIN {X 0,Y 521.715,Z 508.238,A -85,B 0,C 180,E1 22501.977,E2 22501.977} C_VEL
LIN {X 0,Y 521.719,Z 508.218,A -85,B 0,C 180,E1 22498.462,E2 22498.462} C_VEL
LIN {X 0,Y 521.746,Z 508.221,A -85,B 0,C 180,E1 22495.053,E2 22495.053} C_VEL
LIN {X 0,Y 521.72,Z 508.241,A -85,B 0,C 180,E1 22491.625,E2 22491.625} C_VEL
LIN {X 0,Y 521.719,Z 508.237,A -85,B 0,C 180,E1 22488.054,E2 22488.054} C_VEL
LIN {X 0,Y 521.745,Z 508.216,A -85,B 0,C 180,E1 22484.665,E2 22484.665} C_VEL
LIN {X 0,Y 521.728,Z 508.218,A -85,B 0,C 180,E1 22481.212,E2 22481.212} C_VEL
LIN {X 0,Y 521.719,Z 508.225,A -85,B 0,C 180,E1 22477.699,E2 22477.699} C_VEL
LIN {X 0,Y 521.745,Z 508.229,A -85,B 0,C 180,E1 22474.249,E2 22474.249} C_VEL
LIN {X 0,Y 521.745,Z 508.232,A -85,B 0,C 180,E1 22470.745,E2 22470.745} C_VEL
LIN {X 0,Y 521.722,Z 508.231,A -85,B 0,C 180,E1 22467.28,E2 22467.28} C_VEL
LIN {X 0,Y 521.753,Z 508.295,A -85,B 0,C 180,E1 22463.782,E2 22463.782} C_VEL
LIN {X 0,Y 521.838,Z 508.838,A -85,B 0,C 180,E1 22463.559,E2 22463.559} C_VEL
LIN {X 0,Y 523.501,Z 512.332,A -85,B 0,C 180,E1 22462.874,E2 22462.874} C_VEL
LIN {X 0,Y 528.582,Z 522.729,A -85,B 0,C 180,E1 22460.956,E2 22460.956} C_VEL
LIN {X 0,Y 535.468,Z 537.295,A -85,B 0,C 180,E1 22458.478,E2 22458.478} C_VEL
LIN {X 0,Y 543.487,Z 555.934,A -85,B 0,C 180,E1 22455.644,E2 22455.644} C_VEL
LIN {X 0,Y 551.023,Z 575.254,A -85,B 0,C 180,E1 22453.005,E2 22453.005} C_VEL
LIN {X 0,Y 553.466,Z 582.658,A -85,B 0,C 180,E1 22452.084,E2 22452.084} C_VEL
LIN {X 0,Y 548.397,Z 626.017,A -85,B 0,C 180,E1 22448.642,E2 22448.642} C_VEL
LIN {X 0,Y 547.861,Z 632.948,A -85,B 0,C 180,E1 22448.136,E2 22448.136} C_VEL
LIN {X 0,Y 556.852,Z 686.343,A -85,B 0,C 180,E1 22446.487,E2 22446.487} C_VEL
LIN {X 0,Y 557.618,Z 692.598,A -85,B 0,C 180,E1 22446.327,E2 22446.327} C_VEL
LIN {X 0,Y 552.584,Z 943.921,A -85,B 0,C 180,E1 22443.072,E2 22443.072} C_VEL
LIN {X 0,Y 551.463,Z 951.591,A -85,B 0,C 180,E1 22443.026,E2 22443.026} C_VEL
LIN {X 0,Y 545.509,Z 970.825,A -85,B 0,C 180,E1 22443.037,E2 22443.037} C_VEL
LIN {X 0,Y 544.25,Z 978.381,A -85,B 0,C 180,E1 22442.905,E2 22442.905} C_VEL
LIN {X 0,Y 542.309,Z 1000.342,A -85,B 0,C 180,E1 22442.238,E2 22442.238} C_VEL
LIN {X 0,Y 540.184,Z 1020.128,A -85,B 0,C 180,E1 22441.464,E2 22441.464} C_VEL
LIN {X 0,Y 537.629,Z 1039.509,A -85,B 0,C 180,E1 22440.512,E2 22440.512} C_VEL
LIN {X 0,Y 534.715,Z 1059.333,A -85,B 0,C 180,E1 22439.335,E2 22439.335} C_VEL
LIN {X 0,Y 531.769,Z 1077.477,A -85,B 0,C 180,E1 22438.038,E2 22438.038} C_VEL
LIN {X 0,Y 528.611,Z 1095.447,A -85,B 0,C 180,E1 22436.512,E2 22436.512} C_VEL
LIN {X 0,Y 525.596,Z 1112.017,A -85,B 0,C 180,E1 22434.861,E2 22434.861} C_VEL
LIN {X 0,Y 522.731,Z 1127.273,A -85,B 0,C 180,E1 22433.063,E2 22433.063} C_VEL
LIN {X 0,Y 520.044,Z 1141.681,A -85,B 0,C 180,E1 22431.072,E2 22431.072} C_VEL
LIN {X 0,Y 517.811,Z 1154.234,A -85,B 0,C 180,E1 22429.046,E2 22429.046} C_VEL
LIN {X 0,Y 515.838,Z 1165.91,A -85,B 0,C 180,E1 22426.787,E2 22426.787} C_VEL
LIN {X 0,Y 514.309,Z 1176.16,A -85,B 0,C 180,E1 22424.409,E2 22424.409} C_VEL
LIN {X 0,Y 513.25,Z 1184.601,A -85,B 0,C 180,E1 22422.031,E2 22422.031} C_VEL
LIN {X 0,Y 512.579,Z 1191.225,A -85,B 0,C 180,E1 22419.657,E2 22419.657} C_VEL
LIN {X 0,Y 512.169,Z 1196.736,A -85,B 0,C 180,E1 22417.065,E2 22417.065} C_VEL
LIN {X 0,Y 512.011,Z 1200.416,A -85,B 0,C 180,E1 22414.592,E2 22414.592} C_VEL
LIN {X 0,Y 511.955,Z 1202.42,A -85,B 0,C 180,E1 22412.127,E2 22412.127} C_VEL
LIN {X 0,Y 511.936,Z 1202.994,A -85,B 0,C 180,E1 22409.552,E2 22409.552} C_VEL
LIN {X 0,Y 511.96,Z 1202.091,A -85,B 0,C 180,E1 22407.201,E2 22407.201} C_VEL
LIN {X 0,Y 512.031,Z 1199.643,A -85,B 0,C 180,E1 22404.734,E2 22404.734} C_VEL
LIN {X 0,Y 512.244,Z 1195.72,A -85,B 0,C 180,E1 22402.26,E2 22402.26} C_VEL
LIN {X 0,Y 512.686,Z 1190.026,A -85,B 0,C 180,E1 22399.778,E2 22399.778} C_VEL
LIN {X 0,Y 513.472,Z 1182.642,A -85,B 0,C 180,E1 22397.289,E2 22397.289} C_VEL
LIN {X 0,Y 514.649,Z 1173.881,A -85,B 0,C 180,E1 22394.91,E2 22394.91} C_VEL
LIN {X 0,Y 516.218,Z 1163.607,A -85,B 0,C 180,E1 22392.646,E2 22392.646} C_VEL
LIN {X 0,Y 518.295,Z 1151.423,A -85,B 0,C 180,E1 22390.387,E2 22390.387} C_VEL
LIN {X 0,Y 520.653,Z 1138.529,A -85,B 0,C 180,E1 22388.358,E2 22388.358} C_VEL
LIN {X 0,Y 523.311,Z 1124.235,A -85,B 0,C 180,E1 22386.464,E2 22386.464} C_VEL
LIN {X 0,Y 526.416,Z 1107.584,A -85,B 0,C 180,E1 22384.58,E2 22384.58} C_VEL
LIN {X 0,Y 529.456,Z 1091.056,A -85,B 0,C 180,E1 22382.988,E2 22382.988} C_VEL
LIN {X 0,Y 532.428,Z 1073.586,A -85,B 0,C 180,E1 22381.572,E2 22381.572} C_VEL
LIN {X 0,Y 535.502,Z 1054.418,A -85,B 0,C 180,E1 22380.256,E2 22380.256} C_VEL
LIN {X 0,Y 538.14,Z 1036.096,A -85,B 0,C 180,E1 22379.211,E2 22379.211} C_VEL
LIN {X 0,Y 540.753,Z 1015.155,A -85,B 0,C 180,E1 22378.234,E2 22378.234} C_VEL
LIN {X 0,Y 542.948,Z 994.329,A -85,B 0,C 180,E1 22377.457,E2 22377.457} C_VEL
LIN {X 0,Y 544.691,Z 972.851,A -85,B 0,C 180,E1 22376.865,E2 22376.865} C_VEL
LIN {X 0,Y 545.998,Z 949.592,A -85,B 0,C 180,E1 22376.419,E2 22376.419} C_VEL
LIN {X 0,Y 551.469,Z 692.333,A -85,B 0,C 180,E1 22373.032,E2 22373.032} C_VEL
LIN {X 0,Y 542.84,Z 640.022,A -85,B 0,C 180,E1 22371.405,E2 22371.405} C_VEL
LIN {X 0,Y 541.371,Z 631.161,A -85,B 0,C 180,E1 22371.101,E2 22371.101} C_VEL
LIN {X 0,Y 546.511,Z 588.382,A -85,B 0,C 180,E1 22367.68,E2 22367.68} C_VEL
LIN {X 0,Y 546.744,Z 585.338,A -85,B 0,C 180,E1 22367.419,E2 22367.419} C_VEL
LIN {X 0,Y 539.709,Z 566.61,A -85,B 0,C 180,E1 22364.899,E2 22364.899} C_VEL
LIN {X 0,Y 532.344,Z 548.84,A -85,B 0,C 180,E1 22362.255,E2 22362.255} C_VEL
LIN {X 0,Y 525.779,Z 534.298,A -85,B 0,C 180,E1 22359.858,E2 22359.858} C_VEL
LIN {X 0,Y 519.7,Z 521.65,A -85,B 0,C 180,E1 22357.566,E2 22357.566} C_VEL
LIN {X 0,Y 517.344,Z 517.082,A -85,B 0,C 180,E1 22356.671,E2 22356.671} C_VEL
LIN {X 0,Y 515.358,Z 513.024,A -85,B 0,C 180,E1 22355.869,E2 22355.869} C_VEL
LIN {X 0,Y 513.806,Z 509.392,A -85,B 0,C 180,E1 22355.105,E2 22355.105} C_VEL
LIN {X 0,Y 513.811,Z 509.231,A -85,B 0,C 180,E1 22351.697,E2 22351.697} C_VEL
LIN {X 0,Y 513.783,Z 509.234,A -85,B 0,C 180,E1 22348.35,E2 22348.35} C_VEL
LIN {X 0,Y 513.783,Z 509.232,A -85,B 0,C 180,E1 22344.858,E2 22344.858} C_VEL
LIN {X 0,Y 513.813,Z 509.223,A -85,B 0,C 180,E1 22341.46,E2 22341.46} C_VEL
LIN {X 0,Y 513.78,Z 509.214,A -85,B 0,C 180,E1 22338.025,E2 22338.025} C_VEL
LIN {X 0,Y 513.777,Z 509.205,A -85,B 0,C 180,E1 22334.54,E2 22334.54} C_VEL
LIN {X 0,Y 513.807,Z 509.206,A -85,B 0,C 180,E1 22331.108,E2 22331.108} C_VEL
LIN {X 0,Y 513.778,Z 509.233,A -85,B 0,C 180,E1 22327.717,E2 22327.717} C_VEL
LIN {X 0,Y 513.773,Z 509.228,A -85,B 0,C 180,E1 22324.129,E2 22324.129} C_VEL
LIN {X 0,Y 513.811,Z 509.203,A -85,B 0,C 180,E1 22320.669,E2 22320.669} C_VEL
LIN {X 0,Y 513.785,Z 509.209,A -85,B 0,C 180,E1 22317.211,E2 22317.211} C_VEL
LIN {X 0,Y 513.77,Z 509.232,A -85,B 0,C 180,E1 22313.743,E2 22313.743} C_VEL
LIN {X 0,Y 513.807,Z 509.221,A -85,B 0,C 180,E1 22310.366,E2 22310.366} C_VEL
LIN {X 0,Y 513.783,Z 509.206,A -85,B 0,C 180,E1 22306.953,E2 22306.953} C_VEL
LIN {X 0,Y 513.764,Z 509.21,A -85,B 0,C 180,E1 22303.492,E2 22303.492} C_VEL
LIN {X 0,Y 513.806,Z 509.214,A -85,B 0,C 180,E1 22300.036,E2 22300.036} C_VEL
LIN {X 0,Y 513.784,Z 509.226,A -85,B 0,C 180,E1 22296.608,E2 22296.608} C_VEL
LIN {X 0,Y 513.766,Z 509.235,A -85,B 0,C 180,E1 22293.159,E2 22293.159} C_VEL
LIN {X 0,Y 513.816,Z 509.229,A -85,B 0,C 180,E1 22289.768,E2 22289.768} C_VEL
LIN {X 0,Y 513.772,Z 509.152,A -85,B 0,C 180,E1 22286.313,E2 22286.313} C_VEL
LIN {X 0,Y 513.81,Z 509.467,A -85,B 0,C 180,E1 22285.237,E2 22285.237} C_VEL
LIN {X 0,Y 515.267,Z 512.966,A -85,B 0,C 180,E1 22284.534,E2 22284.534} C_VEL
LIN {X 0,Y 516.48,Z 515.17,A -85,B 0,C 180,E1 22284.084,E2 22284.084} C_VEL
LIN {X 0,Y 522.61,Z 527.06,A -85,B 0,C 180,E1 22281.831,E2 22281.831} C_VEL
LIN {X 0,Y 530.465,Z 543.828,A -85,B 0,C 180,E1 22279.008,E2 22279.008} C_VEL
LIN {X 0,Y 533.357,Z 550.18,A -85,B 0,C 180,E1 22278.061,E2 22278.061} C_VEL
LIN {X 0,Y 547.333,Z 571.129,A -85,B 0,C 180,E1 22276.236,E2 22276.236} C_VEL
LIN {X 0,Y 557.948,Z 588.537,A -85,B 0,C 180,E1 22274.923,E2 22274.923} C_VEL
LIN {X 0,Y 550.063,Z 827.201,A -85,B 0,C 180,E1 22271.364,E2 22271.364} C_VEL
LIN {X 0,Y 546.912,Z 923.139,A -85,B 0,C 180,E1 22269.903,E2 22269.903} C_VEL
LIN {X 0,Y 545.363,Z 947.978,A -85,B 0,C 180,E1 22269.352,E2 22269.352} C_VEL
LIN {X 0,Y 543.592,Z 970.21,A -85,B 0,C 180,E1 22268.697,E2 22268.697} C_VEL
LIN {X 0,Y 541.326,Z 993.493,A -85,B 0,C 180,E1 22267.823,E2 22267.823} C_VEL
LIN {X 0,Y 539.006,Z 1014.223,A -85,B 0,C 180,E1 22266.877,E2 22266.877} C_VEL
LIN {X 0,Y 536.035,Z 1037.884,A -85,B 0,C 180,E1 22265.581,E2 22265.581} C_VEL
LIN {X 0,Y 533.305,Z 1057.698,A -85,B 0,C 180,E1 22264.302,E2 22264.302} C_VEL
LIN {X 0,Y 530.116,Z 1079.638,A -85,B 0,C 180,E1 22262.645,E2 22262.645} C_VEL
LIN {X 0,Y 527.355,Z 1097.962,A -85,B 0,C 180,E1 22261.045,E2 22261.045} C_VEL
LIN {X 0,Y 524.349,Z 1117.329,A -85,B 0,C 180,E1 22259.094,E2 22259.094} C_VEL
LIN {X 0,Y 521.849,Z 1133.822,A -85,B 0,C 180,E1 22257.191,E2 22257.191} C_VEL
LIN {X 0,Y 519.325,Z 1150.772,A -85,B 0,C 180,E1 22254.938,E2 22254.938} C_VEL
LIN {X 0,Y 517.415,Z 1164.471,A -85,B 0,C 180,E1 22252.856,E2 22252.856} C_VEL
LIN {X 0,Y 515.618,Z 1178.287,A -85,B 0,C 180,E1 22250.429,E2 22250.429} C_VEL
LIN {X 0,Y 514.393,Z 1189.083,A -85,B 0,C 180,E1 22248.237,E2 22248.237} C_VEL
LIN {X 0,Y 513.272,Z 1200.612,A -85,B 0,C 180,E1 22245.478,E2 22245.478} C_VEL
LIN {X 0,Y 512.662,Z 1208.569,A -85,B 0,C 180,E1 22243.19,E2 22243.19} C_VEL
LIN {X 0,Y 512.203,Z 1216.315,A -85,B 0,C 180,E1 22240.46,E2 22240.46} C_VEL
LIN {X 0,Y 512.013,Z 1221.492,A -85,B 0,C 180,E1 22238.083,E2 22238.083} C_VEL
LIN {X 0,Y 511.926,Z 1225.538,A -85,B 0,C 180,E1 22235.604,E2 22235.604} C_VEL
LIN {X 0,Y 511.902,Z 1228.084,A -85,B 0,C 180,E1 22233.023,E2 22233.023} C_VEL
LIN {X 0,Y 511.908,Z 1229.046,A -85,B 0,C 180,E1 22230.895,E2 22230.895} C_VEL
LIN {X 0,Y 511.919,Z 1228.951,A -85,B 0,C 180,E1 22228.657,E2 22228.657} C_VEL
LIN {X 0,Y 511.93,Z 1227.154,A -85,B 0,C 180,E1 22225.856,E2 22225.856} C_VEL
LIN {X 0,Y 511.966,Z 1224.199,A -85,B 0,C 180,E1 22223.496,E2 22223.496} C_VEL
LIN {X 0,Y 512.08,Z 1219.515,A -85,B 0,C 180,E1 22220.9,E2 22220.9} C_VEL
LIN {X 0,Y 512.353,Z 1213.298,A -85,B 0,C 180,E1 22218.404,E2 22218.404} C_VEL
LIN {X 0,Y 512.811,Z 1206.344,A -85,B 0,C 180,E1 22216.124,E2 22216.124} C_VEL
LIN {X 0,Y 513.639,Z 1196.557,A -85,B 0,C 180,E1 22213.489,E2 22213.489} C_VEL
LIN {X 0,Y 514.626,Z 1186.931,A -85,B 0,C 180,E1 22211.302,E2 22211.302} C_VEL
LIN {X 0,Y 516.105,Z 1174.603,A -85,B 0,C 180,E1 22208.879,E2 22208.879} C_VEL
LIN {X 0,Y 517.796,Z 1161.542,A -85,B 0,C 180,E1 22206.681,E2 22206.681} C_VEL
LIN {X 0,Y 520.039,Z 1146.028,A -85,B 0,C 180,E1 22204.39,E2 22204.39} C_VEL
LIN {X 0,Y 522.405,Z 1129.958,A -85,B 0,C 180,E1 22202.346,E2 22202.346} C_VEL
LIN {X 0,Y 525.207,Z 1111.957,A -85,B 0,C 180,E1 22200.332,E2 22200.332} C_VEL
LIN {X 0,Y 527.991,Z 1093.589,A -85,B 0,C 180,E1 22198.559,E2 22198.559} C_VEL
LIN {X 0,Y 530.961,Z 1073.995,A -85,B 0,C 180,E1 22196.9,E2 22196.9} C_VEL
LIN {X 0,Y 533.872,Z 1053.63,A -85,B 0,C 180,E1 22195.426,E2 22195.426} C_VEL
LIN {X 0,Y 536.817,Z 1032.061,A -85,B 0,C 180,E1 22194.076,E2 22194.076} C_VEL
LIN {X 0,Y 539.387,Z 1010.683,A -85,B 0,C 180,E1 22192.955,E2 22192.955} C_VEL
LIN {X 0,Y 541.942,Z 987.372,A -85,B 0,C 180,E1 22191.926,E2 22191.926} C_VEL
LIN {X 0,Y 544.039,Z 964.18,A -85,B 0,C 180,E1 22191.112,E2 22191.112} C_VEL
LIN {X 0,Y 545.953,Z 939.408,A -85,B 0,C 180,E1 22190.438,E2 22190.438} C_VEL
LIN {X 0,Y 547.183,Z 916.419,A -85,B 0,C 180,E1 22189.988,E2 22189.988} C_VEL
LIN {X 0,Y 555.114,Z 671.863,A -85,B 0,C 180,E1 22186.313,E2 22186.313} C_VEL
LIN {X 0,Y 557.784,Z 588.16,A -85,B 0,C 180,E1 22185.061,E2 22185.061} C_VEL
LIN {X 0,Y 543.926,Z 565.955,A -85,B 0,C 180,E1 22183.344,E2 22183.344} C_VEL
LIN {X 0,Y 533.029,Z 549.668,A -85,B 0,C 180,E1 22181.898,E2 22181.898} C_VEL
LIN {X 0,Y 526.25,Z 534.772,A -85,B 0,C 180,E1 22179.522,E2 22179.522} C_VEL
LIN {X 0,Y 520.026,Z 522.168,A -85,B 0,C 180,E1 22177.277,E2 22177.277} C_VEL
LIN {X 0,Y 517.272,Z 516.9,A -85,B 0,C 180,E1 22176.264,E2 22176.264} C_VEL
LIN {X 0,Y 515.547,Z 513.344,A -85,B 0,C 180,E1 22175.58,E2 22175.58} C_VEL
LIN {X 0,Y 513.846,Z 509.68,A -85,B 0,C 180,E1 22174.846,E2 22174.846} C_VEL
LIN {X 0,Y 513.801,Z 509.152,A -85,B 0,C 180,E1 22174.088,E2 22174.088} C_VEL
LIN {X 0,Y 513.778,Z 509.219,A -85,B 0,C 180,E1 22170.657,E2 22170.657} C_VEL
LIN {X 0,Y 513.77,Z 509.227,A -85,B 0,C 180,E1 22167.205,E2 22167.205} C_VEL
LIN {X 0,Y 513.812,Z 509.216,A -85,B 0,C 180,E1 22163.755,E2 22163.755} C_VEL
LIN {X 0,Y 513.776,Z 509.212,A -85,B 0,C 180,E1 22160.387,E2 22160.387} C_VEL
LIN {X 0,Y 513.768,Z 509.209,A -85,B 0,C 180,E1 22156.857,E2 22156.857} C_VEL
LIN {X 0,Y 513.81,Z 509.21,A -85,B 0,C 180,E1 22153.505,E2 22153.505} C_VEL
LIN {X 0,Y 513.784,Z 509.23,A -85,B 0,C 180,E1 22150.033,E2 22150.033} C_VEL
LIN {X 0,Y 513.774,Z 509.222,A -85,B 0,C 180,E1 22146.593,E2 22146.593} C_VEL
LIN {X 0,Y 513.804,Z 509.201,A -85,B 0,C 180,E1 22143.124,E2 22143.124} C_VEL
LIN {X 0,Y 513.79,Z 509.21,A -85,B 0,C 180,E1 22139.665,E2 22139.665} C_VEL
LIN {X 0,Y 513.775,Z 509.231,A -85,B 0,C 180,E1 22136.206,E2 22136.206} C_VEL
LIN {X 0,Y 513.814,Z 509.217,A -85,B 0,C 180,E1 22132.733,E2 22132.733} C_VEL
LIN {X 0,Y 513.799,Z 509.202,A -85,B 0,C 180,E1 22129.232,E2 22129.232} C_VEL
LIN {X 0,Y 513.773,Z 509.209,A -85,B 0,C 180,E1 22125.805,E2 22125.805} C_VEL
LIN {X 0,Y 513.805,Z 509.22,A -85,B 0,C 180,E1 22122.327,E2 22122.327} C_VEL
LIN {X 0,Y 513.812,Z 509.229,A -85,B 0,C 180,E1 22118.767,E2 22118.767} C_VEL
LIN {X 0,Y 513.781,Z 509.233,A -85,B 0,C 180,E1 22115.265,E2 22115.265} C_VEL
LIN {X 0,Y 513.798,Z 509.228,A -85,B 0,C 180,E1 22111.777,E2 22111.777} C_VEL
LIN {X 0,Y 513.809,Z 509.23,A -85,B 0,C 180,E1 22108.303,E2 22108.303} C_VEL
LIN {X 0,Y 513.81,Z 509.359,A -85,B 0,C 180,E1 22104.798,E2 22104.798} C_VEL
LIN {X 0,Y 515.064,Z 512.613,A -85,B 0,C 180,E1 22104.107,E2 22104.107} C_VEL
LIN {X 0,Y 516.285,Z 514.742,A -85,B 0,C 180,E1 22103.656,E2 22103.656} C_VEL
LIN {X 0,Y 520.717,Z 523.697,A -85,B 0,C 180,E1 22101.93,E2 22101.93} C_VEL
LIN {X 0,Y 526.75,Z 536.462,A -85,B 0,C 180,E1 22099.662,E2 22099.662} C_VEL
LIN {X 0,Y 533.37,Z 551.24,A -85,B 0,C 180,E1 22097.263,E2 22097.263} C_VEL
LIN {X 0,Y 540.772,Z 569.344,A -85,B 0,C 180,E1 22094.613,E2 22094.613} C_VEL
LIN {X 0,Y 546.805,Z 585.758,A -85,B 0,C 180,E1 22092.433,E2 22092.433} C_VEL
LIN {X 0,Y 541.531,Z 629.055,A -85,B 0,C 180,E1 22088.96,E2 22088.96} C_VEL
LIN {X 0,Y 541.467,Z 632.387,A -85,B 0,C 180,E1 22088.75,E2 22088.75} C_VEL
LIN {X 0,Y 550.411,Z 685.887,A -85,B 0,C 180,E1 22087.059,E2 22087.059} C_VEL
LIN {X 0,Y 551.455,Z 693.958,A -85,B 0,C 180,E1 22086.842,E2 22086.842} C_VEL
LIN {X 0,Y 545.846,Z 952.805,A -85,B 0,C 180,E1 22083.439,E2 22083.439} C_VEL
LIN {X 0,Y 544.489,Z 975.002,A -85,B 0,C 180,E1 22082.988,E2 22082.988} C_VEL
LIN {X 0,Y 544.25,Z 978.381,A -85,B 0,C 180,E1 22082.905,E2 22082.905} C_VEL
LIN {X 0,Y 542.881,Z 985.916,A -85,B 0,C 180,E1 22082.766,E2 22082.766} C_VEL
LIN {X 0,Y 536.137,Z 1004.75,A -85,B 0,C 180,E1 22082.518,E2 22082.518} C_VEL
LIN {X 0,Y 534.476,Z 1011.995,A -85,B 0,C 180,E1 22082.294,E2 22082.294} C_VEL
LIN {X 0,Y 531.942,Z 1032.31,A -85,B 0,C 180,E1 22081.376,E2 22081.376} C_VEL
LIN {X 0,Y 529.119,Z 1051.452,A -85,B 0,C 180,E1 22080.301,E2 22080.301} C_VEL
LIN {X 0,Y 525.947,Z 1070.863,A -85,B 0,C 180,E1 22078.997,E2 22078.997} C_VEL
LIN {X 0,Y 522.797,Z 1088.644,A -85,B 0,C 180,E1 22077.57,E2 22077.57} C_VEL
LIN {X 0,Y 519.602,Z 1105.553,A -85,B 0,C 180,E1 22075.962,E2 22075.962} C_VEL
LIN {X 0,Y 516.578,Z 1121.218,A -85,B 0,C 180,E1 22074.226,E2 22074.226} C_VEL
LIN {X 0,Y 513.694,Z 1135.85,A -85,B 0,C 180,E1 22072.306,E2 22072.306} C_VEL
LIN {X 0,Y 511.006,Z 1149.854,A -85,B 0,C 180,E1 22070.143,E2 22070.143} C_VEL
LIN {X 0,Y 508.848,Z 1161.808,A -85,B 0,C 180,E1 22067.969,E2 22067.969} C_VEL
LIN {X 0,Y 507.09,Z 1172.29,A -85,B 0,C 180,E1 22065.672,E2 22065.672} C_VEL
LIN {X 0,Y 505.762,Z 1181.423,A -85,B 0,C 180,E1 22063.257,E2 22063.257} C_VEL
LIN {X 0,Y 504.879,Z 1189.002,A -85,B 0,C 180,E1 22060.792,E2 22060.792} C_VEL
LIN {X 0,Y 504.345,Z 1194.789,A -85,B 0,C 180,E1 22058.321,E2 22058.321} C_VEL
LIN {X 0,Y 504.067,Z 1199.28,A -85,B 0,C 180,E1 22055.692,E2 22055.692} C_VEL
LIN {X 0,Y 503.97,Z 1202.021,A -85,B 0,C 180,E1 22053.184,E2 22053.184} C_VEL
LIN {X 0,Y 503.945,Z 1203.138,A -85,B 0,C 180,E1 22050.682,E2 22050.682} C_VEL
LIN {X 0,Y 503.951,Z 1202.87,A -85,B 0,C 180,E1 22048.181,E2 22048.181} C_VEL
LIN {X 0,Y 503.998,Z 1201.148,A -85,B 0,C 180,E1 22045.791,E2 22045.791} C_VEL
LIN {X 0,Y 504.149,Z 1197.699,A -85,B 0,C 180,E1 22043.166,E2 22043.166} C_VEL
LIN {X 0,Y 504.518,Z 1192.822,A -85,B 0,C 180,E1 22040.648,E2 22040.648} C_VEL
LIN {X 0,Y 505.186,Z 1186.124,A -85,B 0,C 180,E1 22038.122,E2 22038.122} C_VEL
LIN {X 0,Y 506.291,Z 1177.65,A -85,B 0,C 180,E1 22035.592,E2 22035.592} C_VEL
LIN {X 0,Y 507.842,Z 1167.735,A -85,B 0,C 180,E1 22033.177,E2 22033.177} C_VEL
LIN {X 0,Y 509.832,Z 1156.246,A -85,B 0,C 180,E1 22030.882,E2 22030.882} C_VEL
LIN {X 0,Y 512.251,Z 1143.355,A -85,B 0,C 180,E1 22028.712,E2 22028.712} C_VEL
LIN {X 0,Y 514.879,Z 1129.968,A -85,B 0,C 180,E1 22026.783,E2 22026.783} C_VEL
LIN {X 0,Y 517.758,Z 1115.171,A -85,B 0,C 180,E1 22024.981,E2 22024.981} C_VEL
LIN {X 0,Y 521.055,Z 1098.047,A -85,B 0,C 180,E1 22023.196,E2 22023.196} C_VEL
LIN {X 0,Y 524.182,Z 1081.193,A -85,B 0,C 180,E1 22021.706,E2 22021.706} C_VEL
LIN {X 0,Y 527.32,Z 1062.81,A -85,B 0,C 180,E1 22020.338,E2 22020.338} C_VEL
LIN {X 0,Y 530.32,Z 1043.838,A -85,B 0,C 180,E1 22019.148,E2 22019.148} C_VEL
LIN {X 0,Y 532.909,Z 1025.071,A -85,B 0,C 180,E1 22018.182,E2 22018.182} C_VEL
LIN {X 0,Y 535.488,Z 1003.38,A -85,B 0,C 180,E1 22017.279,E2 22017.279} C_VEL
LIN {X 0,Y 537.461,Z 983.023,A -85,B 0,C 180,E1 22016.62,E2 22016.62} C_VEL
LIN {X 0,Y 539.017,Z 961.22,A -85,B 0,C 180,E1 22016.111,E2 22016.111} C_VEL
LIN {X 0,Y 539.987,Z 936.868,A -85,B 0,C 180,E1 22015.726,E2 22015.726} C_VEL
LIN {X 0,Y 545.352,Z 693.727,A -85,B 0,C 180,E1 22012.505,E2 22012.505} C_VEL
LIN {X 0,Y 536.669,Z 640.294,A -85,B 0,C 180,E1 22010.811,E2 22010.811} C_VEL
LIN {X 0,Y 534.992,Z 630.018,A -85,B 0,C 180,E1 22010.444,E2 22010.444} C_VEL
LIN {X 0,Y 540.167,Z 589.236,A -85,B 0,C 180,E1 22007.141,E2 22007.141} C_VEL
LIN {X 0,Y 533.422,Z 571.071,A -85,B 0,C 180,E1 22004.663,E2 22004.663} C_VEL
LIN {X 0,Y 525.834,Z 552.619,A -85,B 0,C 180,E1 22001.87,E2 22001.87} C_VEL
LIN {X 0,Y 519.635,Z 538.917,A -85,B 0,C 180,E1 21999.562,E2 21999.562} C_VEL
LIN {X 0,Y 513.973,Z 526.982,A -85,B 0,C 180,E1 21997.371,E2 21997.371} C_VEL
LIN {X 0,Y 509.842,Z 518.674,A -85,B 0,C 180,E1 21995.718,E2 21995.718} C_VEL
LIN {X 0,Y 507.45,Z 514.125,A -85,B 0,C 180,E1 21994.751,E2 21994.751} C_VEL
LIN {X 0,Y 505.892,Z 510.37,A -85,B 0,C 180,E1 21993.933,E2 21993.933} C_VEL
LIN {X 0,Y 505.844,Z 510.201,A -85,B 0,C 180,E1 21990.4,E2 21990.4} C_VEL
LIN {X 0,Y 505.845,Z 510.198,A -85,B 0,C 180,E1 21986.915,E2 21986.915} C_VEL
LIN {X 0,Y 505.871,Z 510.194,A -85,B 0,C 180,E1 21983.409,E2 21983.409} C_VEL
LIN {X 0,Y 505.847,Z 510.203,A -85,B 0,C 180,E1 21979.997,E2 21979.997} C_VEL
LIN {X 0,Y 505.836,Z 510.219,A -85,B 0,C 180,E1 21976.42,E2 21976.42} C_VEL
LIN {X 0,Y 505.871,Z 510.216,A -85,B 0,C 180,E1 21972.988,E2 21972.988} C_VEL
LIN {X 0,Y 505.858,Z 510.197,A -85,B 0,C 180,E1 21969.443,E2 21969.443} C_VEL
LIN {X 0,Y 505.83,Z 510.194,A -85,B 0,C 180,E1 21966.014,E2 21966.014} C_VEL
LIN {X 0,Y 505.855,Z 510.209,A -85,B 0,C 180,E1 21962.492,E2 21962.492} C_VEL
LIN {X 0,Y 505.872,Z 510.219,A -85,B 0,C 180,E1 21958.981,E2 21958.981} C_VEL
LIN {X 0,Y 505.83,Z 510.203,A -85,B 0,C 180,E1 21955.465,E2 21955.465} C_VEL
LIN {X 0,Y 505.836,Z 510.191,A -85,B 0,C 180,E1 21951.932,E2 21951.932} C_VEL
LIN {X 0,Y 505.87,Z 510.201,A -85,B 0,C 180,E1 21948.484,E2 21948.484} C_VEL
LIN {X 0,Y 505.83,Z 510.223,A -85,B 0,C 180,E1 21945.109,E2 21945.109} C_VEL
LIN {X 0,Y 505.835,Z 510.217,A -85,B 0,C 180,E1 21941.562,E2 21941.562} C_VEL
LIN {X 0,Y 505.877,Z 510.199,A -85,B 0,C 180,E1 21938.064,E2 21938.064} C_VEL
LIN {X 0,Y 505.84,Z 510.2,A -85,B 0,C 180,E1 21934.598,E2 21934.598} C_VEL
LIN {X 0,Y 505.822,Z 510.204,A -85,B 0,C 180,E1 21931.125,E2 21931.125} C_VEL
LIN {X 0,Y 505.866,Z 510.147,A -85,B 0,C 180,E1 21927.879,E2 21927.879} C_VEL
LIN {X 0,Y 505.867,Z 510.43,A -85,B 0,C 180,E1 21926.43,E2 21926.43} C_VEL
LIN {X 0,Y 507.649,Z 514.317,A -85,B 0,C 180,E1 21925.577,E2 21925.577} C_VEL
LIN {X 0,Y 511.083,Z 521.09,A -85,B 0,C 180,E1 21924.199,E2 21924.199} C_VEL
LIN {X 0,Y 517.131,Z 533.063,A -85,B 0,C 180,E1 21921.917,E2 21921.917} C_VEL
LIN {X 0,Y 523.319,Z 546.399,A -85,B 0,C 180,E1 21919.63,E2 21919.63} C_VEL
LIN {X 0,Y 525.795,Z 551.437,A -85,B 0,C 180,E1 21918.854,E2 21918.854} C_VEL
LIN {X 0,Y 539.035,Z 571.114,A -85,B 0,C 180,E1 21917.059,E2 21917.059} C_VEL
LIN {X 0,Y 551.852,Z 591.723,A -85,B 0,C 180,E1 21915.429,E2 21915.429} C_VEL
LIN {X 0,Y 543.782,Z 826.961,A -85,B 0,C 180,E1 21911.888,E2 21911.888} C_VEL
LIN {X 0,Y 540.489,Z 923.409,A -85,B 0,C 180,E1 21910.405,E2 21910.405} C_VEL
LIN {X 0,Y 538.879,Z 948.311,A -85,B 0,C 180,E1 21909.848,E2 21909.848} C_VEL
LIN {X 0,Y 537.023,Z 970.762,A -85,B 0,C 180,E1 21909.179,E2 21909.179} C_VEL
LIN {X 0,Y 534.699,Z 993.688,A -85,B 0,C 180,E1 21908.308,E2 21908.308} C_VEL
LIN {X 0,Y 532.289,Z 1014.401,A -85,B 0,C 180,E1 21907.353,E2 21907.353} C_VEL
LIN {X 0,Y 529.16,Z 1038.328,A -85,B 0,C 180,E1 21906.027,E2 21906.027} C_VEL
LIN {X 0,Y 526.338,Z 1057.978,A -85,B 0,C 180,E1 21904.743,E2 21904.743} C_VEL
LIN {X 0,Y 523.024,Z 1079.729,A -85,B 0,C 180,E1 21903.078,E2 21903.078} C_VEL
LIN {X 0,Y 520.14,Z 1098.032,A -85,B 0,C 180,E1 21901.46,E2 21901.46} C_VEL
LIN {X 0,Y 517.049,Z 1117.099,A -85,B 0,C 180,E1 21899.514,E2 21899.514} C_VEL
LIN {X 0,Y 514.509,Z 1132.88,A -85,B 0,C 180,E1 21897.675,E2 21897.675} C_VEL
LIN {X 0,Y 511.789,Z 1150.36,A -85,B 0,C 180,E1 21895.331,E2 21895.331} C_VEL
LIN {X 0,Y 509.756,Z 1164.077,A -85,B 0,C 180,E1 21893.219,E2 21893.219} C_VEL
LIN {X 0,Y 507.846,Z 1178.032,A -85,B 0,C 180,E1 21890.736,E2 21890.736} C_VEL
LIN {X 0,Y 506.557,Z 1188.741,A -85,B 0,C 180,E1 21888.529,E2 21888.529} C_VEL
LIN {X 0,Y 505.406,Z 1199.878,A -85,B 0,C 180,E1 21885.843,E2 21885.843} C_VEL
LIN {X 0,Y 504.739,Z 1207.904,A -85,B 0,C 180,E1 21883.518,E2 21883.518} C_VEL
LIN {X 0,Y 504.278,Z 1215.239,A -85,B 0,C 180,E1 21880.973,E2 21880.973} C_VEL
LIN {X 0,Y 504.041,Z 1221.026,A -85,B 0,C 180,E1 21878.326,E2 21878.326} C_VEL
LIN {X 0,Y 503.948,Z 1224.97,A -85,B 0,C 180,E1 21875.922,E2 21875.922} C_VEL
LIN {X 0,Y 503.91,Z 1227.8,A -85,B 0,C 180,E1 21873.185,E2 21873.185} C_VEL
LIN {X 0,Y 503.911,Z 1228.841,A -85,B 0,C 180,E1 21870.91,E2 21870.91} C_VEL
LIN {X 0,Y 503.92,Z 1228.745,A -85,B 0,C 180,E1 21868.636,E2 21868.636} C_VEL
LIN {X 0,Y 503.932,Z 1226.934,A -85,B 0,C 180,E1 21865.79,E2 21865.79} C_VEL
LIN {X 0,Y 503.97,Z 1223.964,A -85,B 0,C 180,E1 21863.392,E2 21863.392} C_VEL
LIN {X 0,Y 504.094,Z 1219.252,A -85,B 0,C 180,E1 21860.755,E2 21860.755} C_VEL
LIN {X 0,Y 504.385,Z 1213.018,A -85,B 0,C 180,E1 21858.219,E2 21858.219} C_VEL
LIN {X 0,Y 504.9,Z 1205.677,A -85,B 0,C 180,E1 21855.785,E2 21855.785} C_VEL
LIN {X 0,Y 505.8,Z 1195.75,A -85,B 0,C 180,E1 21853.107,E2 21853.107} C_VEL
LIN {X 0,Y 506.861,Z 1186.05,A -85,B 0,C 180,E1 21850.885,E2 21850.885} C_VEL
LIN {X 0,Y 508.539,Z 1172.9,A -85,B 0,C 180,E1 21848.307,E2 21848.307} C_VEL
LIN {X 0,Y 510.281,Z 1160.418,A -85,B 0,C 180,E1 21846.194,E2 21846.194} C_VEL
LIN {X 0,Y 512.771,Z 1143.928,A -85,B 0,C 180,E1 21843.766,E2 21843.766} C_VEL
LIN {X 0,Y 515.255,Z 1128.261,A -85,B 0,C 180,E1 21841.766,E2 21841.766} C_VEL
LIN {X 0,Y 518.32,Z 1109.13,A -85,B 0,C 180,E1 21839.642,E2 21839.642} C_VEL
LIN {X 0,Y 521.118,Z 1091.709,A -85,B 0,C 180,E1 21837.96,E2 21837.96} C_VEL
LIN {X 0,Y 524.475,Z 1070.316,A -85,B 0,C 180,E1 21836.174,E2 21836.174} C_VEL
LIN {X 0,Y 527.324,Z 1051.253,A -85,B 0,C 180,E1 21834.801,E2 21834.801} C_VEL
LIN {X 0,Y 530.497,Z 1028.102,A -85,B 0,C 180,E1 21833.379,E2 21833.379} C_VEL
LIN {X 0,Y 533.107,Z 1007.402,A -85,B 0,C 180,E1 21832.308,E2 21832.308} C_VEL
LIN {X 0,Y 535.768,Z 983.088,A -85,B 0,C 180,E1 21831.27,E2 21831.27} C_VEL
LIN {X 0,Y 537.841,Z 961.009,A -85,B 0,C 180,E1 21830.512,E2 21830.512} C_VEL
LIN {X 0,Y 539.719,Z 936.188,A -85,B 0,C 180,E1 21829.864,E2 21829.864} C_VEL
LIN {X 0,Y 540.891,Z 913.905,A -85,B 0,C 180,E1 21829.438,E2 21829.438} C_VEL
LIN {X 0,Y 549.152,Z 668.164,A -85,B 0,C 180,E1 21825.716,E2 21825.716} C_VEL
LIN {X 0,Y 551.697,Z 591.498,A -85,B 0,C 180,E1 21824.559,E2 21824.559} C_VEL
LIN {X 0,Y 537.648,Z 568.943,A -85,B 0,C 180,E1 21822.769,E2 21822.769} C_VEL
LIN {X 0,Y 525.254,Z 550.528,A -85,B 0,C 180,E1 21821.053,E2 21821.053} C_VEL
LIN {X 0,Y 518.607,Z 536.194,A -85,B 0,C 180,E1 21818.659,E2 21818.659} C_VEL
LIN {X 0,Y 513.979,Z 526.918,A -85,B 0,C 180,E1 21816.951,E2 21816.951} C_VEL
LIN {X 0,Y 510.192,Z 519.188,A -85,B 0,C 180,E1 21815.459,E2 21815.459} C_VEL
LIN {X 0,Y 507.275,Z 513.787,A -85,B 0,C 180,E1 21814.324,E2 21814.324} C_VEL
LIN {X 0,Y 505.864,Z 510.386,A -85,B 0,C 180,E1 21813.57,E2 21813.57} C_VEL
LIN {X 0,Y 505.854,Z 510.212,A -85,B 0,C 180,E1 21810.482,E2 21810.482} C_VEL
LIN {X 0,Y 505.829,Z 510.219,A -85,B 0,C 180,E1 21807.043,E2 21807.043} C_VEL
LIN {X 0,Y 505.86,Z 510.21,A -85,B 0,C 180,E1 21803.533,E2 21803.533} C_VEL
LIN {X 0,Y 505.858,Z 510.201,A -85,B 0,C 180,E1 21800.117,E2 21800.117} C_VEL
LIN {X 0,Y 505.827,Z 510.197,A -85,B 0,C 180,E1 21796.656,E2 21796.656} C_VEL
LIN {X 0,Y 505.861,Z 510.195,A -85,B 0,C 180,E1 21793.255,E2 21793.255} C_VEL
LIN {X 0,Y 505.861,Z 510.214,A -85,B 0,C 180,E1 21789.787,E2 21789.787} C_VEL
LIN {X 0,Y 505.832,Z 510.217,A -85,B 0,C 180,E1 21786.355,E2 21786.355} C_VEL
LIN {X 0,Y 505.853,Z 510.193,A -85,B 0,C 180,E1 21782.832,E2 21782.832} C_VEL
LIN {X 0,Y 505.87,Z 510.192,A -85,B 0,C 180,E1 21779.434,E2 21779.434} C_VEL
LIN {X 0,Y 505.835,Z 510.218,A -85,B 0,C 180,E1 21775.919,E2 21775.919} C_VEL
LIN {X 0,Y 505.851,Z 510.216,A -85,B 0,C 180,E1 21772.39,E2 21772.39} C_VEL
LIN {X 0,Y 505.868,Z 510.192,A -85,B 0,C 180,E1 21768.946,E2 21768.946} C_VEL
LIN {X 0,Y 505.836,Z 510.195,A -85,B 0,C 180,E1 21765.578,E2 21765.578} C_VEL
LIN {X 0,Y 505.852,Z 510.205,A -85,B 0,C 180,E1 21762.04,E2 21762.04} C_VEL
LIN {X 0,Y 505.872,Z 510.215,A -85,B 0,C 180,E1 21758.551,E2 21758.551} C_VEL
LIN {X 0,Y 505.849,Z 510.221,A -85,B 0,C 180,E1 21755.1,E2 21755.1} C_VEL
LIN {X 0,Y 505.847,Z 510.224,A -85,B 0,C 180,E1 21751.551,E2 21751.551} C_VEL
LIN {X 0,Y 505.871,Z 510.221,A -85,B 0,C 180,E1 21748.147,E2 21748.147} C_VEL
LIN {X 0,Y 505.903,Z 510.462,A -85,B 0,C 180,E1 21745.904,E2 21745.904} C_VEL
LIN {X 0,Y 507.392,Z 514.041,A -85,B 0,C 180,E1 21745.146,E2 21745.146} C_VEL
LIN {X 0,Y 508.542,Z 516.166,A -85,B 0,C 180,E1 21744.686,E2 21744.686} C_VEL
LIN {X 0,Y 510.849,Z 520.744,A -85,B 0,C 180,E1 21743.744,E2 21743.744} C_VEL
LIN {X 0,Y 514.925,Z 528.852,A -85,B 0,C 180,E1 21742.148,E2 21742.148} C_VEL
LIN {X 0,Y 521.021,Z 541.936,A -85,B 0,C 180,E1 21739.798,E2 21739.798} C_VEL
LIN {X 0,Y 527.784,Z 557.235,A -85,B 0,C 180,E1 21737.294,E2 21737.294} C_VEL
LIN {X 0,Y 535.016,Z 575.238,A -85,B 0,C 180,E1 21734.642,E2 21734.642} C_VEL
LIN {X 0,Y 540.11,Z 589.278,A -85,B 0,C 180,E1 21732.757,E2 21732.757} C_VEL
LIN {X 0,Y 534.965,Z 630.603,A -85,B 0,C 180,E1 21729.425,E2 21729.425} C_VEL
LIN {X 0,Y 543.976,Z 685.138,A -85,B 0,C 180,E1 21727.654,E2 21727.654} C_VEL
LIN {X 0,Y 545.335,Z 695.371,A -85,B 0,C 180,E1 21727.368,E2 21727.368} C_VEL
LIN {X 0,Y 539.451,Z 952.625,A -85,B 0,C 180,E1 21723.95,E2 21723.95} C_VEL
LIN {X 0,Y 538.039,Z 974.882,A -85,B 0,C 180,E1 21723.495,E2 21723.495} C_VEL
LIN {X 0,Y 536.229,Z 995.891,A -85,B 0,C 180,E1 21722.893,E2 21722.893} C_VEL
LIN {X 0,Y 534.476,Z 1011.995,A -85,B 0,C 180,E1 21722.294,E2 21722.294} C_VEL
LIN {X 0,Y 532.773,Z 1019.472,A -85,B 0,C 180,E1 21722.046,E2 21722.046} C_VEL
LIN {X 0,Y 525.357,Z 1037.374,A -85,B 0,C 180,E1 21721.539,E2 21721.539} C_VEL
LIN {X 0,Y 523.513,Z 1044.256,A -85,B 0,C 180,E1 21721.223,E2 21721.223} C_VEL
LIN {X 0,Y 520.423,Z 1062.987,A -85,B 0,C 180,E1 21720.032,E2 21720.032} C_VEL
LIN {X 0,Y 517.062,Z 1081.875,A -85,B 0,C 180,E1 21718.604,E2 21718.604} C_VEL
LIN {X 0,Y 513.811,Z 1098.772,A -85,B 0,C 180,E1 21717.088,E2 21717.088} C_VEL
LIN {X 0,Y 510.481,Z 1115.324,A -85,B 0,C 180,E1 21715.334,E2 21715.334} C_VEL
LIN {X 0,Y 507.4,Z 1130.49,A -85,B 0,C 180,E1 21713.456,E2 21713.456} C_VEL
LIN {X 0,Y 504.664,Z 1143.839,A -85,B 0,C 180,E1 21711.502,E2 21711.502} C_VEL
LIN {X 0,Y 502.02,Z 1157.276,A -85,B 0,C 180,E1 21709.185,E2 21709.185} C_VEL
LIN {X 0,Y 499.966,Z 1168.626,A -85,B 0,C 180,E1 21706.857,E2 21706.857} C_VEL
LIN {X 0,Y 498.366,Z 1178.432,A -85,B 0,C 180,E1 21704.405,E2 21704.405} C_VEL
LIN {X 0,Y 497.223,Z 1186.76,A -85,B 0,C 180,E1 21701.836,E2 21701.836} C_VEL
LIN {X 0,Y 496.533,Z 1193.33,A -85,B 0,C 180,E1 21699.27,E2 21699.27} C_VEL
LIN {X 0,Y 496.155,Z 1198.147,A -85,B 0,C 180,E1 21696.712,E2 21696.712} C_VEL
LIN {X 0,Y 495.998,Z 1201.481,A -85,B 0,C 180,E1 21694.046,E2 21694.046} C_VEL
LIN {X 0,Y 495.946,Z 1203.195,A -85,B 0,C 180,E1 21691.502,E2 21691.502} C_VEL
LIN {X 0,Y 495.947,Z 1203.296,A -85,B 0,C 180,E1 21688.96,E2 21688.96} C_VEL
LIN {X 0,Y 495.984,Z 1201.885,A -85,B 0,C 180,E1 21686.297,E2 21686.297} C_VEL
LIN {X 0,Y 496.099,Z 1199.165,A -85,B 0,C 180,E1 21683.868,E2 21683.868} C_VEL
LIN {X 0,Y 496.409,Z 1194.726,A -85,B 0,C 180,E1 21681.311,E2 21681.311} C_VEL
LIN {X 0,Y 497.009,Z 1188.709,A -85,B 0,C 180,E1 21678.747,E2 21678.747} C_VEL
LIN {X 0,Y 497.959,Z 1181.21,A -85,B 0,C 180,E1 21676.294,E2 21676.294} C_VEL
LIN {X 0,Y 499.394,Z 1171.966,A -85,B 0,C 180,E1 21673.841,E2 21673.841} C_VEL
LIN {X 0,Y 501.276,Z 1161.411,A -85,B 0,C 180,E1 21671.51,E2 21671.51} C_VEL
LIN {X 0,Y 503.641,Z 1149.006,A -85,B 0,C 180,E1 21669.243,E2 21669.243} C_VEL
LIN {X 0,Y 506.424,Z 1135.215,A -85,B 0,C 180,E1 21667.111,E2 21667.111} C_VEL
LIN {X 0,Y 509.479,Z 1120.482,A -85,B 0,C 180,E1 21665.167,E2 21665.167} C_VEL
LIN {X 0,Y 512.677,Z 1104.563,A -85,B 0,C 180,E1 21663.398,E2 21663.398} C_VEL
LIN {X 0,Y 516.249,Z 1086.265,A -85,B 0,C 180,E1 21661.673,E2 21661.673} C_VEL
LIN {X 0,Y 519.594,Z 1068.204,A -85,B 0,C 180,E1 21660.233,E2 21660.233} C_VEL
LIN {X 0,Y 522.625,Z 1049.971,A -85,B 0,C 180,E1 21659.027,E2 21659.027} C_VEL
LIN {X 0,Y 525.705,Z 1029.325,A -85,B 0,C 180,E1 21657.887,E2 21657.887} C_VEL
LIN {X 0,Y 528.2,Z 1010.114,A -85,B 0,C 180,E1 21657.028,E2 21657.028} C_VEL
LIN {X 0,Y 530.466,Z 988.765,A -85,B 0,C 180,E1 21656.279,E2 21656.279} C_VEL
LIN {X 0,Y 532.276,Z 967.446,A -85,B 0,C 180,E1 21655.716,E2 21655.716} C_VEL
LIN {X 0,Y 533.413,Z 945.241,A -85,B 0,C 180,E1 21655.321,E2 21655.321} C_VEL
LIN {X 0,Y 539.267,Z 695.06,A -85,B 0,C 180,E1 21651.964,E2 21651.964} C_VEL
LIN {X 0,Y 530.801,Z 642.18,A -85,B 0,C 180,E1 21650.257,E2 21650.257} C_VEL
LIN {X 0,Y 528.687,Z 628.878,A -85,B 0,C 180,E1 21649.771,E2 21649.771} C_VEL
LIN {X 0,Y 533.493,Z 592.76,A -85,B 0,C 180,E1 21646.809,E2 21646.809} C_VEL
LIN {X 0,Y 526.829,Z 574.723,A -85,B 0,C 180,E1 21644.302,E2 21644.302} C_VEL
LIN {X 0,Y 519.336,Z 556.427,A -85,B 0,C 180,E1 21641.477,E2 21641.477} C_VEL
LIN {X 0,Y 512.683,Z 541.446,A -85,B 0,C 180,E1 21638.903,E2 21638.903} C_VEL
LIN {X 0,Y 506.498,Z 528.694,A -85,B 0,C 180,E1 21636.457,E2 21636.457} C_VEL
LIN {X 0,Y 501.97,Z 519.807,A -85,B 0,C 180,E1 21634.59,E2 21634.59} C_VEL
LIN {X 0,Y 499.843,Z 515.478,A -85,B 0,C 180,E1 21633.65,E2 21633.65} C_VEL
LIN {X 0,Y 498.028,Z 511.937,A -85,B 0,C 180,E1 21632.825,E2 21632.825} C_VEL
LIN {X 0,Y 497.913,Z 511.276,A -85,B 0,C 180,E1 21632.561,E2 21632.561} C_VEL
LIN {X 0,Y 497.906,Z 511.203,A -85,B 0,C 180,E1 21628.945,E2 21628.945} C_VEL
LIN {X 0,Y 497.932,Z 511.197,A -85,B 0,C 180,E1 21625.451,E2 21625.451} C_VEL
LIN {X 0,Y 497.919,Z 511.191,A -85,B 0,C 180,E1 21621.917,E2 21621.917} C_VEL
LIN {X 0,Y 497.896,Z 511.186,A -85,B 0,C 180,E1 21618.379,E2 21618.379} C_VEL
LIN {X 0,Y 497.925,Z 511.178,A -85,B 0,C 180,E1 21614.895,E2 21614.895} C_VEL
LIN {X 0,Y 497.926,Z 511.186,A -85,B 0,C 180,E1 21611.35,E2 21611.35} C_VEL
LIN {X 0,Y 497.896,Z 511.212,A -85,B 0,C 180,E1 21607.849,E2 21607.849} C_VEL
LIN {X 0,Y 497.901,Z 511.202,A -85,B 0,C 180,E1 21604.261,E2 21604.261} C_VEL
LIN {X 0,Y 497.933,Z 511.178,A -85,B 0,C 180,E1 21600.805,E2 21600.805} C_VEL
LIN {X 0,Y 497.899,Z 511.188,A -85,B 0,C 180,E1 21597.353,E2 21597.353} C_VEL
LIN {X 0,Y 497.893,Z 511.21,A -85,B 0,C 180,E1 21593.744,E2 21593.744} C_VEL
LIN {X 0,Y 497.926,Z 511.199,A -85,B 0,C 180,E1 21590.289,E2 21590.289} C_VEL
LIN {X 0,Y 497.918,Z 511.183,A -85,B 0,C 180,E1 21586.766,E2 21586.766} C_VEL
LIN {X 0,Y 497.884,Z 511.185,A -85,B 0,C 180,E1 21583.31,E2 21583.31} C_VEL
LIN {X 0,Y 497.911,Z 511.188,A -85,B 0,C 180,E1 21579.793,E2 21579.793} C_VEL
LIN {X 0,Y 497.93,Z 511.193,A -85,B 0,C 180,E1 21576.299,E2 21576.299} C_VEL
LIN {X 0,Y 497.89,Z 511.204,A -85,B 0,C 180,E1 21572.826,E2 21572.826} C_VEL
LIN {X 0,Y 497.89,Z 511.184,A -85,B 0,C 180,E1 21569.196,E2 21569.196} C_VEL
LIN {X 0,Y 497.956,Z 511.392,A -85,B 0,C 180,E1 21567.685,E2 21567.685} C_VEL
LIN {X 0,Y 499.456,Z 515.002,A -85,B 0,C 180,E1 21566.87,E2 21566.87} C_VEL
LIN {X 0,Y 500.677,Z 517.112,A -85,B 0,C 180,E1 21566.382,E2 21566.382} C_VEL
LIN {X 0,Y 503.364,Z 522.515,A -85,B 0,C 180,E1 21565.242,E2 21565.242} C_VEL
LIN {X 0,Y 505.701,Z 526.982,A -85,B 0,C 180,E1 21564.318,E2 21564.318} C_VEL
LIN {X 0,Y 511.4,Z 538.327,A -85,B 0,C 180,E1 21562.125,E2 21562.125} C_VEL
LIN {X 0,Y 517.679,Z 551.959,A -85,B 0,C 180,E1 21559.771,E2 21559.771} C_VEL
LIN {X 0,Y 531.235,Z 571.782,A -85,B 0,C 180,E1 21557.855,E2 21557.855} C_VEL
LIN {X 0,Y 544.725,Z 593.124,A -85,B 0,C 180,E1 21556.082,E2 21556.082} C_VEL
LIN {X 0,Y 545.8,Z 595.432,A -85,B 0,C 180,E1 21555.936,E2 21555.936} C_VEL
LIN {X 0,Y 537.308,Z 833.822,A -85,B 0,C 180,E1 21552.316,E2 21552.316} C_VEL
LIN {X 0,Y 534.106,Z 923.79,A -85,B 0,C 180,E1 21550.918,E2 21550.918} C_VEL
LIN {X 0,Y 532.443,Z 948.59,A -85,B 0,C 180,E1 21550.357,E2 21550.357} C_VEL
LIN {X 0,Y 530.505,Z 971.227,A -85,B 0,C 180,E1 21549.676,E2 21549.676} C_VEL
LIN {X 0,Y 528.113,Z 993.902,A -85,B 0,C 180,E1 21548.805,E2 21548.805} C_VEL
LIN {X 0,Y 525.614,Z 1014.595,A -85,B 0,C 180,E1 21547.842,E2 21547.842} C_VEL
LIN {X 0,Y 522.431,Z 1038.078,A -85,B 0,C 180,E1 21546.527,E2 21546.527} C_VEL
LIN {X 0,Y 519.557,Z 1057.289,A -85,B 0,C 180,E1 21545.263,E2 21545.263} C_VEL
LIN {X 0,Y 516.074,Z 1079.187,A -85,B 0,C 180,E1 21543.579,E2 21543.579} C_VEL
LIN {X 0,Y 513.056,Z 1097.492,A -85,B 0,C 180,E1 21541.945,E2 21541.945} C_VEL
LIN {X 0,Y 509.777,Z 1116.9,A -85,B 0,C 180,E1 21539.945,E2 21539.945} C_VEL
LIN {X 0,Y 507.063,Z 1132.916,A -85,B 0,C 180,E1 21538.053,E2 21538.053} C_VEL
LIN {X 0,Y 504.276,Z 1149.967,A -85,B 0,C 180,E1 21535.736,E2 21535.736} C_VEL
LIN {X 0,Y 502.123,Z 1163.701,A -85,B 0,C 180,E1 21533.593,E2 21533.593} C_VEL
LIN {X 0,Y 500.036,Z 1178.191,A -85,B 0,C 180,E1 21530.973,E2 21530.973} C_VEL
LIN {X 0,Y 498.67,Z 1188.956,A -85,B 0,C 180,E1 21528.712,E2 21528.712} C_VEL
LIN {X 0,Y 497.464,Z 1200.009,A -85,B 0,C 180,E1 21525.983,E2 21525.983} C_VEL
LIN {X 0,Y 496.765,Z 1207.996,A -85,B 0,C 180,E1 21523.62,E2 21523.62} C_VEL
LIN {X 0,Y 496.271,Z 1215.53,A -85,B 0,C 180,E1 21520.917,E2 21520.917} C_VEL
LIN {X 0,Y 496.055,Z 1220.787,A -85,B 0,C 180,E1 21518.461,E2 21518.461} C_VEL
LIN {X 0,Y 495.953,Z 1224.746,A -85,B 0,C 180,E1 21516.018,E2 21516.018} C_VEL
LIN {X 0,Y 495.914,Z 1227.591,A -85,B 0,C 180,E1 21513.236,E2 21513.236} C_VEL
LIN {X 0,Y 495.914,Z 1228.636,A -85,B 0,C 180,E1 21510.924,E2 21510.924} C_VEL
LIN {X 0,Y 495.922,Z 1228.54,A -85,B 0,C 180,E1 21508.614,E2 21508.614} C_VEL
LIN {X 0,Y 495.933,Z 1226.838,A -85,B 0,C 180,E1 21505.838,E2 21505.838} C_VEL
LIN {X 0,Y 495.97,Z 1223.904,A -85,B 0,C 180,E1 21503.402,E2 21503.402} C_VEL
LIN {X 0,Y 496.097,Z 1219.259,A -85,B 0,C 180,E1 21500.721,E2 21500.721} C_VEL
LIN {X 0,Y 496.399,Z 1213.071,A -85,B 0,C 180,E1 21498.144,E2 21498.144} C_VEL
LIN {X 0,Y 496.902,Z 1206.137,A -85,B 0,C 180,E1 21495.789,E2 21495.789} C_VEL
LIN {X 0,Y 497.877,Z 1195.918,A -85,B 0,C 180,E1 21492.95,E2 21492.95} C_VEL
LIN {X 0,Y 498.986,Z 1186.262,A -85,B 0,C 180,E1 21490.693,E2 21490.693} C_VEL
LIN {X 0,Y 500.743,Z 1173.2,A -85,B 0,C 180,E1 21488.075,E2 21488.075} C_VEL
LIN {X 0,Y 502.684,Z 1160.039,A -85,B 0,C 180,E1 21485.811,E2 21485.811} C_VEL
LIN {X 0,Y 505.349,Z 1143.242,A -85,B 0,C 180,E1 21483.312,E2 21483.312} C_VEL
LIN {X 0,Y 507.971,Z 1127.612,A -85,B 0,C 180,E1 21481.297,E2 21481.297} C_VEL
LIN {X 0,Y 511.15,Z 1108.622,A -85,B 0,C 180,E1 21479.17,E2 21479.17} C_VEL
LIN {X 0,Y 514.076,Z 1091.263,A -85,B 0,C 180,E1 21477.477,E2 21477.477} C_VEL
LIN {X 0,Y 517.524,Z 1070.18,A -85,B 0,C 180,E1 21475.702,E2 21475.702} C_VEL
LIN {X 0,Y 520.435,Z 1051.472,A -85,B 0,C 180,E1 21474.339,E2 21474.339} C_VEL
LIN {X 0,Y 523.748,Z 1028.267,A -85,B 0,C 180,E1 21472.897,E2 21472.897} C_VEL
LIN {X 0,Y 526.464,Z 1007.591,A -85,B 0,C 180,E1 21471.816,E2 21471.816} C_VEL
LIN {X 0,Y 529.219,Z 983.38,A -85,B 0,C 180,E1 21470.773,E2 21470.773} C_VEL
LIN {X 0,Y 531.363,Z 961.361,A -85,B 0,C 180,E1 21470.01,E2 21470.01} C_VEL
LIN {X 0,Y 533.314,Z 936.428,A -85,B 0,C 180,E1 21469.352,E2 21469.352} C_VEL
LIN {X 0,Y 534.523,Z 914.173,A -85,B 0,C 180,E1 21468.922,E2 21468.922} C_VEL
LIN {X 0,Y 543.092,Z 668.869,A -85,B 0,C 180,E1 21465.172,E2 21465.172} C_VEL
LIN {X 0,Y 545.644,Z 594.719,A -85,B 0,C 180,E1 21464.044,E2 21464.044} C_VEL
LIN {X 0,Y 532.194,Z 573.283,A -85,B 0,C 180,E1 21462.287,E2 21462.287} C_VEL
LIN {X 0,Y 519.363,Z 554.359,A -85,B 0,C 180,E1 21460.506,E2 21460.506} C_VEL
LIN {X 0,Y 517.505,Z 551.612,A -85,B 0,C 180,E1 21460.191,E2 21460.191} C_VEL
LIN {X 0,Y 511.06,Z 537.571,A -85,B 0,C 180,E1 21457.762,E2 21457.762} C_VEL
LIN {X 0,Y 504.497,Z 524.556,A -85,B 0,C 180,E1 21455.222,E2 21455.222} C_VEL
LIN {X 0,Y 501.614,Z 519.11,A -85,B 0,C 180,E1 21454.065,E2 21454.065} C_VEL
LIN {X 0,Y 499.663,Z 515.266,A -85,B 0,C 180,E1 21453.234,E2 21453.234} C_VEL
LIN {X 0,Y 497.997,Z 511.668,A -85,B 0,C 180,E1 21452.435,E2 21452.435} C_VEL
LIN {X 0,Y 497.909,Z 511.145,A -85,B 0,C 180,E1 21451.745,E2 21451.745} C_VEL
LIN {X 0,Y 497.913,Z 511.187,A -85,B 0,C 180,E1 21448.412,E2 21448.412} C_VEL
LIN {X 0,Y 497.886,Z 511.188,A -85,B 0,C 180,E1 21444.944,E2 21444.944} C_VEL
LIN {X 0,Y 497.918,Z 511.185,A -85,B 0,C 180,E1 21441.437,E2 21441.437} C_VEL
LIN {X 0,Y 497.927,Z 511.19,A -85,B 0,C 180,E1 21437.893,E2 21437.893} C_VEL
LIN {X 0,Y 497.892,Z 511.21,A -85,B 0,C 180,E1 21434.42,E2 21434.42} C_VEL
LIN {X 0,Y 497.903,Z 511.204,A -85,B 0,C 180,E1 21430.881,E2 21430.881} C_VEL
LIN {X 0,Y 497.932,Z 511.177,A -85,B 0,C 180,E1 21427.384,E2 21427.384} C_VEL
LIN {X 0,Y 497.901,Z 511.18,A -85,B 0,C 180,E1 21423.915,E2 21423.915} C_VEL
LIN {X 0,Y 497.896,Z 511.201,A -85,B 0,C 180,E1 21420.345,E2 21420.345} C_VEL
LIN {X 0,Y 497.929,Z 511.204,A -85,B 0,C 180,E1 21416.892,E2 21416.892} C_VEL
LIN {X 0,Y 497.927,Z 511.184,A -85,B 0,C 180,E1 21413.312,E2 21413.312} C_VEL
LIN {X 0,Y 497.895,Z 511.18,A -85,B 0,C 180,E1 21409.821,E2 21409.821} C_VEL
LIN {X 0,Y 497.92,Z 511.19,A -85,B 0,C 180,E1 21406.293,E2 21406.293} C_VEL
LIN {X 0,Y 497.933,Z 511.205,A -85,B 0,C 180,E1 21402.711,E2 21402.711} C_VEL
LIN {X 0,Y 497.913,Z 511.209,A -85,B 0,C 180,E1 21399.179,E2 21399.179} C_VEL
LIN {X 0,Y 497.907,Z 511.199,A -85,B 0,C 180,E1 21395.69,E2 21395.69} C_VEL
LIN {X 0,Y 497.934,Z 511.195,A -85,B 0,C 180,E1 21392.103,E2 21392.103} C_VEL
LIN {X 0,Y 497.933,Z 511.2,A -85,B 0,C 180,E1 21388.526,E2 21388.526} C_VEL
LIN {X 0,Y 497.953,Z 511.531,A -85,B 0,C 180,E1 21387.132,E2 21387.132} C_VEL
LIN {X 0,Y 499.541,Z 515.097,A -85,B 0,C 180,E1 21386.327,E2 21386.327} C_VEL
LIN {X 0,Y 500.639,Z 517.163,A -85,B 0,C 180,E1 21385.859,E2 21385.859} C_VEL
LIN {X 0,Y 503.374,Z 522.62,A -85,B 0,C 180,E1 21384.687,E2 21384.687} C_VEL
LIN {X 0,Y 505.639,Z 527.119,A -85,B 0,C 180,E1 21383.753,E2 21383.753} C_VEL
LIN {X 0,Y 509.708,Z 535.402,A -85,B 0,C 180,E1 21382.12,E2 21382.12} C_VEL
LIN {X 0,Y 515.389,Z 547.624,A -85,B 0,C 180,E1 21379.901,E2 21379.901} C_VEL
LIN {X 0,Y 522.201,Z 563.226,A -85,B 0,C 180,E1 21377.326,E2 21377.326} C_VEL
LIN {X 0,Y 529.457,Z 581.614,A -85,B 0,C 180,E1 21374.604,E2 21374.604} C_VEL
LIN {X 0,Y 533.436,Z 592.615,A -85,B 0,C 180,E1 21373.105,E2 21373.105} C_VEL
LIN {X 0,Y 528.658,Z 629.903,A -85,B 0,C 180,E1 21370.072,E2 21370.072} C_VEL
LIN {X 0,Y 537.739,Z 685.35,A -85,B 0,C 180,E1 21368.234,E2 21368.234} C_VEL
LIN {X 0,Y 539.263,Z 696.768,A -85,B 0,C 180,E1 21367.907,E2 21367.907} C_VEL
LIN {X 0,Y 533.104,Z 952.305,A -85,B 0,C 180,E1 21364.476,E2 21364.476} C_VEL
LIN {X 0,Y 531.653,Z 974.499,A -85,B 0,C 180,E1 21364.019,E2 21364.019} C_VEL
LIN {X 0,Y 529.764,Z 995.639,A -85,B 0,C 180,E1 21363.411,E2 21363.411} C_VEL
LIN {X 0,Y 527.45,Z 1015.84,A -85,B 0,C 180,E1 21362.637,E2 21362.637} C_VEL
LIN {X 0,Y 524.564,Z 1037.129,A -85,B 0,C 180,E1 21361.612,E2 21361.612} C_VEL
LIN {X 0,Y 523.513,Z 1044.256,A -85,B 0,C 180,E1 21361.223,E2 21361.223} C_VEL
LIN {X 0,Y 521.607,Z 1051.109,A -85,B 0,C 180,E1 21360.88,E2 21360.88} C_VEL
LIN {X 0,Y 513.567,Z 1068.188,A -85,B 0,C 180,E1 21360.097,E2 21360.097} C_VEL
LIN {X 0,Y 511.506,Z 1074.551,A -85,B 0,C 180,E1 21359.668,E2 21359.668} C_VEL
LIN {X 0,Y 508.043,Z 1092.462,A -85,B 0,C 180,E1 21358.149,E2 21358.149} C_VEL
LIN {X 0,Y 504.719,Z 1108.577,A -85,B 0,C 180,E1 21356.533,E2 21356.533} C_VEL
LIN {X 0,Y 501.29,Z 1124.652,A -85,B 0,C 180,E1 21354.637,E2 21354.637} C_VEL
LIN {X 0,Y 498.259,Z 1138.966,A -85,B 0,C 180,E1 21352.662,E2 21352.662} C_VEL
LIN {X 0,Y 495.408,Z 1152.5,A -85,B 0,C 180,E1 21350.436,E2 21350.436} C_VEL
LIN {X 0,Y 493.005,Z 1164.566,A -85,B 0,C 180,E1 21348.077,E2 21348.077} C_VEL
LIN {X 0,Y 491.174,Z 1174.752,A -85,B 0,C 180,E1 21345.708,E2 21345.708} C_VEL
LIN {X 0,Y 489.792,Z 1183.459,A -85,B 0,C 180,E1 21343.217,E2 21343.217} C_VEL
LIN {X 0,Y 488.859,Z 1190.77,A -85,B 0,C 180,E1 21340.607,E2 21340.607} C_VEL
LIN {X 0,Y 488.318,Z 1196.417,A -85,B 0,C 180,E1 21338.003,E2 21338.003} C_VEL
LIN {X 0,Y 488.065,Z 1200.306,A -85,B 0,C 180,E1 21335.407,E2 21335.407} C_VEL
LIN {X 0,Y 487.969,Z 1202.783,A -85,B 0,C 180,E1 21332.701,E2 21332.701} C_VEL
LIN {X 0,Y 487.951,Z 1203.654,A -85,B 0,C 180,E1 21330.117,E2 21330.117} C_VEL
LIN {X 0,Y 487.963,Z 1202.962,A -85,B 0,C 180,E1 21327.534,E2 21327.534} C_VEL
LIN {X 0,Y 488.036,Z 1200.879,A -85,B 0,C 180,E1 21324.946,E2 21324.946} C_VEL
LIN {X 0,Y 488.261,Z 1197.157,A -85,B 0,C 180,E1 21322.351,E2 21322.351} C_VEL
LIN {X 0,Y 488.77,Z 1191.576,A -85,B 0,C 180,E1 21319.629,E2 21319.629} C_VEL
LIN {X 0,Y 489.609,Z 1184.914,A -85,B 0,C 180,E1 21317.139,E2 21317.139} C_VEL
LIN {X 0,Y 490.893,Z 1176.408,A -85,B 0,C 180,E1 21314.646,E2 21314.646} C_VEL
LIN {X 0,Y 492.829,Z 1165.545,A -85,B 0,C 180,E1 21312.038,E2 21312.038} C_VEL
LIN {X 0,Y 495.054,Z 1154.373,A -85,B 0,C 180,E1 21309.796,E2 21309.796} C_VEL
LIN {X 0,Y 497.643,Z 1141.776,A -85,B 0,C 180,E1 21307.683,E2 21307.683} C_VEL
LIN {X 0,Y 500.973,Z 1126.245,A -85,B 0,C 180,E1 21305.472,E2 21305.472} C_VEL
LIN {X 0,Y 504.358,Z 1110.492,A -85,B 0,C 180,E1 21303.573,E2 21303.573} C_VEL
LIN {X 0,Y 507.706,Z 1094.223,A -85,B 0,C 180,E1 21301.922,E2 21301.922} C_VEL
LIN {X 0,Y 511.409,Z 1075.257,A -85,B 0,C 180,E1 21300.29,E2 21300.29} C_VEL
LIN {X 0,Y 514.798,Z 1056.76,A -85,B 0,C 180,E1 21298.952,E2 21298.952} C_VEL
LIN {X 0,Y 517.907,Z 1037.43,A -85,B 0,C 180,E1 21297.803,E2 21297.803} C_VEL
LIN {X 0,Y 520.904,Z 1016.254,A -85,B 0,C 180,E1 21296.77,E2 21296.77} C_VEL
LIN {X 0,Y 523.295,Z 996.137,A -85,B 0,C 180,E1 21295.989,E2 21295.989} C_VEL
LIN {X 0,Y 525.319,Z 974.57,A -85,B 0,C 180,E1 21295.358,E2 21295.358} C_VEL
LIN {X 0,Y 526.834,Z 952.451,A -85,B 0,C 180,E1 21294.897,E2 21294.897} C_VEL
LIN {X 0,Y 530.12,Z 820.159,A -85,B 0,C 180,E1 21293.1,E2 21293.1} C_VEL
LIN {X 0,Y 533.177,Z 695.984,A -85,B 0,C 180,E1 21291.398,E2 21291.398} C_VEL
LIN {X 0,Y 524.833,Z 643.096,A -85,B 0,C 180,E1 21289.657,E2 21289.657} C_VEL
LIN {X 0,Y 522.431,Z 628.213,A -85,B 0,C 180,E1 21289.113,E2 21289.113} C_VEL
LIN {X 0,Y 526.798,Z 596.149,A -85,B 0,C 180,E1 21286.452,E2 21286.452} C_VEL
LIN {X 0,Y 519.952,Z 577.559,A -85,B 0,C 180,E1 21283.812,E2 21283.812} C_VEL
LIN {X 0,Y 512.846,Z 560.273,A -85,B 0,C 180,E1 21281.075,E2 21281.075} C_VEL
LIN {X 0,Y 506.569,Z 546.104,A -85,B 0,C 180,E1 21278.59,E2 21278.59} C_VEL
LIN {X 0,Y 500.764,Z 533.978,A -85,B 0,C 180,E1 21276.23,E2 21276.23} C_VEL
LIN {X 0,Y 496.587,Z 525.612,A -85,B 0,C 180,E1 21274.458,E2 21274.458} C_VEL
LIN {X 0,Y 494.152,Z 520.879,A -85,B 0,C 180,E1 21273.393,E2 21273.393} C_VEL
LIN {X 0,Y 491.778,Z 516.343,A -85,B 0,C 180,E1 21272.326,E2 21272.326} C_VEL
LIN {X 0,Y 490.076,Z 512.71,A -85,B 0,C 180,E1 21271.453,E2 21271.453} C_VEL
LIN {X 0,Y 489.966,Z 512.183,A -85,B 0,C 180,E1 21270.949,E2 21270.949} C_VEL
LIN {X 0,Y 489.992,Z 512.176,A -85,B 0,C 180,E1 21267.422,E2 21267.422} C_VEL
LIN {X 0,Y 489.986,Z 512.177,A -85,B 0,C 180,E1 21263.832,E2 21263.832} C_VEL
LIN {X 0,Y 489.96,Z 512.187,A -85,B 0,C 180,E1 21260.3,E2 21260.3} C_VEL
LIN {X 0,Y 489.972,Z 512.197,A -85,B 0,C 180,E1 21256.723,E2 21256.723} C_VEL
LIN {X 0,Y 489.995,Z 512.186,A -85,B 0,C 180,E1 21253.212,E2 21253.212} C_VEL
LIN {X 0,Y 489.968,Z 512.171,A -85,B 0,C 180,E1 21249.633,E2 21249.633} C_VEL
LIN {X 0,Y 489.953,Z 512.171,A -85,B 0,C 180,E1 21246.092,E2 21246.092} C_VEL
LIN {X 0,Y 489.982,Z 512.186,A -85,B 0,C 180,E1 21242.573,E2 21242.573} C_VEL
LIN {X 0,Y 489.99,Z 512.195,A -85,B 0,C 180,E1 21239.065,E2 21239.065} C_VEL
LIN {X 0,Y 489.95,Z 512.177,A -85,B 0,C 180,E1 21235.552,E2 21235.552} C_VEL
LIN {X 0,Y 489.965,Z 512.167,A -85,B 0,C 180,E1 21232.023,E2 21232.023} C_VEL
LIN {X 0,Y 489.992,Z 512.176,A -85,B 0,C 180,E1 21228.464,E2 21228.464} C_VEL
LIN {X 0,Y 489.96,Z 512.199,A -85,B 0,C 180,E1 21224.979,E2 21224.979} C_VEL
LIN {X 0,Y 489.953,Z 512.197,A -85,B 0,C 180,E1 21221.436,E2 21221.436} C_VEL
LIN {X 0,Y 489.988,Z 512.18,A -85,B 0,C 180,E1 21217.883,E2 21217.883} C_VEL
LIN {X 0,Y 489.978,Z 512.177,A -85,B 0,C 180,E1 21214.366,E2 21214.366} C_VEL
LIN {X 0,Y 489.946,Z 512.183,A -85,B 0,C 180,E1 21210.861,E2 21210.861} C_VEL
LIN {X 0,Y 489.993,Z 512.496,A -85,B 0,C 180,E1 21208.985,E2 21208.985} C_VEL
LIN {X 0,Y 491.439,Z 515.845,A -85,B 0,C 180,E1 21208.199,E2 21208.199} C_VEL
LIN {X 0,Y 492.62,Z 517.619,A -85,B 0,C 180,E1 21207.736,E2 21207.736} C_VEL
LIN {X 0,Y 494.466,Z 521.281,A -85,B 0,C 180,E1 21206.908,E2 21206.908} C_VEL
LIN {X 0,Y 498.014,Z 528.381,A -85,B 0,C 180,E1 21205.375,E2 21205.375} C_VEL
LIN {X 0,Y 501.81,Z 535.709,A -85,B 0,C 180,E1 21203.857,E2 21203.857} C_VEL
LIN {X 0,Y 508.136,Z 548.957,A -85,B 0,C 180,E1 21201.368,E2 21201.368} C_VEL
LIN {X 0,Y 510.36,Z 553.639,A -85,B 0,C 180,E1 21200.596,E2 21200.596} C_VEL
LIN {X 0,Y 523.685,Z 572.727,A -85,B 0,C 180,E1 21198.652,E2 21198.652} C_VEL
LIN {X 0,Y 537.225,Z 594.067,A -85,B 0,C 180,E1 21196.807,E2 21196.807} C_VEL
LIN {X 0,Y 539.801,Z 598.687,A -85,B 0,C 180,E1 21196.462,E2 21196.462} C_VEL
LIN {X 0,Y 530.959,Z 838.04,A -85,B 0,C 180,E1 21192.796,E2 21192.796} C_VEL
LIN {X 0,Y 527.77,Z 924.158,A -85,B 0,C 180,E1 21191.444,E2 21191.444} C_VEL
LIN {X 0,Y 526.052,Z 948.878,A -85,B 0,C 180,E1 21190.879,E2 21190.879} C_VEL
LIN {X 0,Y 524.018,Z 971.82,A -85,B 0,C 180,E1 21190.182,E2 21190.182} C_VEL
LIN {X 0,Y 521.57,Z 994.138,A -85,B 0,C 180,E1 21189.314,E2 21189.314} C_VEL
LIN {X 0,Y 518.979,Z 1014.809,A -85,B 0,C 180,E1 21188.342,E2 21188.342} C_VEL
LIN {X 0,Y 515.677,Z 1038.255,A -85,B 0,C 180,E1 21187.016,E2 21187.016} C_VEL
LIN {X 0,Y 512.705,Z 1057.364,A -85,B 0,C 180,E1 21185.744,E2 21185.744} C_VEL
LIN {X 0,Y 508.991,Z 1079.699,A -85,B 0,C 180,E1 21184.003,E2 21184.003} C_VEL
LIN {X 0,Y 505.907,Z 1097.594,A -85,B 0,C 180,E1 21182.384,E2 21182.384} C_VEL
LIN {X 0,Y 502.486,Z 1116.971,A -85,B 0,C 180,E1 21180.359,E2 21180.359} C_VEL
LIN {X 0,Y 499.647,Z 1132.967,A -85,B 0,C 180,E1 21178.442,E2 21178.442} C_VEL
LIN {X 0,Y 496.779,Z 1149.645,A -85,B 0,C 180,E1 21176.144,E2 21176.144} C_VEL
LIN {X 0,Y 494.516,Z 1163.339,A -85,B 0,C 180,E1 21173.979,E2 21173.979} C_VEL
LIN {X 0,Y 492.313,Z 1177.865,A -85,B 0,C 180,E1 21171.318,E2 21171.318} C_VEL
LIN {X 0,Y 490.851,Z 1188.644,A -85,B 0,C 180,E1 21169.021,E2 21169.021} C_VEL
LIN {X 0,Y 489.57,Z 1199.727,A -85,B 0,C 180,E1 21166.248,E2 21166.248} C_VEL
LIN {X 0,Y 488.819,Z 1207.728,A -85,B 0,C 180,E1 21163.846,E2 21163.846} C_VEL
LIN {X 0,Y 488.293,Z 1215.286,A -85,B 0,C 180,E1 21161.098,E2 21161.098} C_VEL
LIN {X 0,Y 488.061,Z 1220.556,A -85,B 0,C 180,E1 21158.601,E2 21158.601} C_VEL
LIN {X 0,Y 487.958,Z 1224.525,A -85,B 0,C 180,E1 21156.117,E2 21156.117} C_VEL
LIN {X 0,Y 487.917,Z 1227.383,A -85,B 0,C 180,E1 21153.289,E2 21153.289} C_VEL
LIN {X 0,Y 487.918,Z 1228.432,A -85,B 0,C 180,E1 21150.939,E2 21150.939} C_VEL
LIN {X 0,Y 487.924,Z 1228.335,A -85,B 0,C 180,E1 21148.591,E2 21148.591} C_VEL
LIN {X 0,Y 487.934,Z 1226.624,A -85,B 0,C 180,E1 21145.769,E2 21145.769} C_VEL
LIN {X 0,Y 487.973,Z 1223.682,A -85,B 0,C 180,E1 21143.293,E2 21143.293} C_VEL
LIN {X 0,Y 488.115,Z 1219.021,A -85,B 0,C 180,E1 21140.568,E2 21140.568} C_VEL
LIN {X 0,Y 488.438,Z 1212.814,A -85,B 0,C 180,E1 21137.948,E2 21137.948} C_VEL
LIN {X 0,Y 488.972,Z 1205.867,A -85,B 0,C 180,E1 21135.554,E2 21135.554} C_VEL
LIN {X 0,Y 490.01,Z 1195.621,A -85,B 0,C 180,E1 21132.668,E2 21132.668} C_VEL
LIN {X 0,Y 491.27,Z 1185.41,A -85,B 0,C 180,E1 21130.254,E2 21130.254} C_VEL
LIN {X 0,Y 493.144,Z 1172.19,A -85,B 0,C 180,E1 21127.594,E2 21127.594} C_VEL
LIN {X 0,Y 495.107,Z 1159.674,A -85,B 0,C 180,E1 21125.417,E2 21125.417} C_VEL
LIN {X 0,Y 497.923,Z 1142.834,A -85,B 0,C 180,E1 21122.882,E2 21122.882} C_VEL
LIN {X 0,Y 500.598,Z 1127.626,A -85,B 0,C 180,E1 21120.894,E2 21120.894} C_VEL
LIN {X 0,Y 503.923,Z 1108.703,A -85,B 0,C 180,E1 21118.745,E2 21118.745} C_VEL
LIN {X 0,Y 506.997,Z 1091.267,A -85,B 0,C 180,E1 21117.023,E2 21117.023} C_VEL
LIN {X 0,Y 510.529,Z 1070.562,A -85,B 0,C 180,E1 21115.256,E2 21115.256} C_VEL
LIN {X 0,Y 513.467,Z 1052.426,A -85,B 0,C 180,E1 21113.915,E2 21113.915} C_VEL
LIN {X 0,Y 516.994,Z 1028.799,A -85,B 0,C 180,E1 21112.422,E2 21112.422} C_VEL
LIN {X 0,Y 519.864,Z 1007.794,A -85,B 0,C 180,E1 21111.312,E2 21111.312} C_VEL
LIN {X 0,Y 522.713,Z 983.68,A -85,B 0,C 180,E1 21110.263,E2 21110.263} C_VEL
LIN {X 0,Y 524.927,Z 961.735,A -85,B 0,C 180,E1 21109.495,E2 21109.495} C_VEL
LIN {X 0,Y 526.955,Z 936.689,A -85,B 0,C 180,E1 21108.827,E2 21108.827} C_VEL
LIN {X 0,Y 528.198,Z 914.54,A -85,B 0,C 180,E1 21108.396,E2 21108.396} C_VEL
LIN {X 0,Y 537.078,Z 669.702,A -85,B 0,C 180,E1 21104.619,E2 21104.619} C_VEL
LIN {X 0,Y 539.639,Z 598.023,A -85,B 0,C 180,E1 21103.518,E2 21103.518} C_VEL
LIN {X 0,Y 525.554,Z 575.587,A -85,B 0,C 180,E1 21101.623,E2 21101.623} C_VEL
LIN {X 0,Y 511.814,Z 555.691,A -85,B 0,C 180,E1 21099.651,E2 21099.651} C_VEL
LIN {X 0,Y 509.856,Z 552.743,A -85,B 0,C 180,E1 21099.305,E2 21099.305} C_VEL
LIN {X 0,Y 503.521,Z 539.157,A -85,B 0,C 180,E1 21096.846,E2 21096.846} C_VEL
LIN {X 0,Y 498.517,Z 529.378,A -85,B 0,C 180,E1 21094.864,E2 21094.864} C_VEL
LIN {X 0,Y 496.163,Z 524.734,A -85,B 0,C 180,E1 21093.875,E2 21093.875} C_VEL
LIN {X 0,Y 494.387,Z 521.171,A -85,B 0,C 180,E1 21093.098,E2 21093.098} C_VEL
LIN {X 0,Y 491.99,Z 516.534,A -85,B 0,C 180,E1 21092.035,E2 21092.035} C_VEL
LIN {X 0,Y 490.143,Z 513.192,A -85,B 0,C 180,E1 21091.209,E2 21091.209} C_VEL
LIN {X 0,Y 489.971,Z 512.341,A -85,B 0,C 180,E1 21090.948,E2 21090.948} C_VEL
LIN {X 0,Y 489.965,Z 512.185,A -85,B 0,C 180,E1 21087.416,E2 21087.416} C_VEL
LIN {X 0,Y 489.996,Z 512.179,A -85,B 0,C 180,E1 21083.831,E2 21083.831} C_VEL
LIN {X 0,Y 489.958,Z 512.176,A -85,B 0,C 180,E1 21080.425,E2 21080.425} C_VEL
LIN {X 0,Y 489.952,Z 512.173,A -85,B 0,C 180,E1 21076.844,E2 21076.844} C_VEL
LIN {X 0,Y 489.992,Z 512.173,A -85,B 0,C 180,E1 21073.452,E2 21073.452} C_VEL
LIN {X 0,Y 489.977,Z 512.193,A -85,B 0,C 180,E1 21069.87,E2 21069.87} C_VEL
LIN {X 0,Y 489.955,Z 512.194,A -85,B 0,C 180,E1 21066.327,E2 21066.327} C_VEL
LIN {X 0,Y 489.973,Z 512.169,A -85,B 0,C 180,E1 21062.807,E2 21062.807} C_VEL
LIN {X 0,Y 489.994,Z 512.166,A -85,B 0,C 180,E1 21059.298,E2 21059.298} C_VEL
LIN {X 0,Y 489.962,Z 512.193,A -85,B 0,C 180,E1 21055.787,E2 21055.787} C_VEL
LIN {X 0,Y 489.962,Z 512.2,A -85,B 0,C 180,E1 21052.141,E2 21052.141} C_VEL
LIN {X 0,Y 489.986,Z 512.175,A -85,B 0,C 180,E1 21048.583,E2 21048.583} C_VEL
LIN {X 0,Y 489.997,Z 512.165,A -85,B 0,C 180,E1 21044.98,E2 21044.98} C_VEL
LIN {X 0,Y 489.964,Z 512.173,A -85,B 0,C 180,E1 21041.436,E2 21041.436} C_VEL
LIN {X 0,Y 489.97,Z 512.179,A -85,B 0,C 180,E1 21037.819,E2 21037.819} C_VEL
LIN {X 0,Y 489.989,Z 512.181,A -85,B 0,C 180,E1 21034.236,E2 21034.236} C_VEL
LIN {X 0,Y 489.995,Z 512.181,A -85,B 0,C 180,E1 21030.611,E2 21030.611} C_VEL
LIN {X 0,Y 490.024,Z 512.404,A -85,B 0,C 180,E1 21028.509,E2 21028.509} C_VEL
LIN {X 0,Y 491.486,Z 515.956,A -85,B 0,C 180,E1 21027.652,E2 21027.652} C_VEL
LIN {X 0,Y 492.649,Z 517.886,A -85,B 0,C 180,E1 21027.165,E2 21027.165} C_VEL
LIN {X 0,Y 495.24,Z 523.017,A -85,B 0,C 180,E1 21025.995,E2 21025.995} C_VEL
LIN {X 0,Y 499.675,Z 531.756,A -85,B 0,C 180,E1 21024.104,E2 21024.104} C_VEL
LIN {X 0,Y 505.718,Z 544.352,A -85,B 0,C 180,E1 21021.623,E2 21021.623} C_VEL
LIN {X 0,Y 512.312,Z 559.012,A -85,B 0,C 180,E1 21019.021,E2 21019.021} C_VEL
LIN {X 0,Y 519.405,Z 576.219,A -85,B 0,C 180,E1 21016.282,E2 21016.282} C_VEL
LIN {X 0,Y 526.402,Z 595.077,A -85,B 0,C 180,E1 21013.59,E2 21013.59} C_VEL
LIN {X 0,Y 526.734,Z 596.594,A -85,B 0,C 180,E1 21013.405,E2 21013.405} C_VEL
LIN {X 0,Y 522.401,Z 628.963,A -85,B 0,C 180,E1 21010.747,E2 21010.747} C_VEL
LIN {X 0,Y 531.518,Z 685.349,A -85,B 0,C 180,E1 21008.835,E2 21008.835} C_VEL
LIN {X 0,Y 533.24,Z 698.137,A -85,B 0,C 180,E1 21008.457,E2 21008.457} C_VEL
LIN {X 0,Y 526.793,Z 952.188,A -85,B 0,C 180,E1 21005.011,E2 21005.011} C_VEL
LIN {X 0,Y 525.287,Z 974.413,A -85,B 0,C 180,E1 21004.549,E2 21004.549} C_VEL
LIN {X 0,Y 523.344,Z 995.372,A -85,B 0,C 180,E1 21003.942,E2 21003.942} C_VEL
LIN {X 0,Y 520.942,Z 1015.591,A -85,B 0,C 180,E1 21003.162,E2 21003.162} C_VEL
LIN {X 0,Y 517.95,Z 1036.914,A -85,B 0,C 180,E1 21002.129,E2 21002.129} C_VEL
LIN {X 0,Y 514.825,Z 1056.391,A -85,B 0,C 180,E1 21000.975,E2 21000.975} C_VEL
LIN {X 0,Y 511.506,Z 1074.551,A -85,B 0,C 180,E1 20999.668,E2 20999.668} C_VEL
LIN {X 0,Y 509.448,Z 1080.94,A -85,B 0,C 180,E1 20999.221,E2 20999.221} C_VEL
LIN {X 0,Y 501.07,Z 1096.703,A -85,B 0,C 180,E1 20998.174,E2 20998.174} C_VEL
LIN {X 0,Y 498.928,Z 1102.519,A -85,B 0,C 180,E1 20997.641,E2 20997.641} C_VEL
LIN {X 0,Y 495.519,Z 1118.047,A -85,B 0,C 180,E1 20995.903,E2 20995.903} C_VEL
LIN {X 0,Y 492.028,Z 1133.627,A -85,B 0,C 180,E1 20993.853,E2 20993.853} C_VEL
LIN {X 0,Y 489.005,Z 1147.41,A -85,B 0,C 180,E1 20991.721,E2 20991.721} C_VEL
LIN {X 0,Y 486.353,Z 1159.687,A -85,B 0,C 180,E1 20989.454,E2 20989.454} C_VEL
LIN {X 0,Y 484.074,Z 1171.124,A -85,B 0,C 180,E1 20986.932,E2 20986.932} C_VEL
LIN {X 0,Y 482.414,Z 1180.619,A -85,B 0,C 180,E1 20984.401,E2 20984.401} C_VEL
LIN {X 0,Y 481.275,Z 1188.238,A -85,B 0,C 180,E1 20981.869,E2 20981.869} C_VEL
LIN {X 0,Y 480.524,Z 1194.735,A -85,B 0,C 180,E1 20979.099,E2 20979.099} C_VEL
LIN {X 0,Y 480.147,Z 1199.316,A -85,B 0,C 180,E1 20976.457,E2 20976.457} C_VEL
LIN {X 0,Y 479.997,Z 1202.218,A -85,B 0,C 180,E1 20973.822,E2 20973.822} C_VEL
LIN {X 0,Y 479.954,Z 1203.688,A -85,B 0,C 180,E1 20971.074,E2 20971.074} C_VEL
LIN {X 0,Y 479.953,Z 1203.642,A -85,B 0,C 180,E1 20968.568,E2 20968.568} C_VEL
LIN {X 0,Y 480.005,Z 1202.091,A -85,B 0,C 180,E1 20965.939,E2 20965.939} C_VEL
LIN {X 0,Y 480.165,Z 1199.124,A -85,B 0,C 180,E1 20963.304,E2 20963.304} C_VEL
LIN {X 0,Y 480.551,Z 1194.446,A -85,B 0,C 180,E1 20960.66,E2 20960.66} C_VEL
LIN {X 0,Y 481.326,Z 1187.834,A -85,B 0,C 180,E1 20957.889,E2 20957.889} C_VEL
LIN {X 0,Y 482.505,Z 1180.147,A -85,B 0,C 180,E1 20955.356,E2 20955.356} C_VEL
LIN {X 0,Y 484.197,Z 1170.52,A -85,B 0,C 180,E1 20952.825,E2 20952.825} C_VEL
LIN {X 0,Y 486.514,Z 1158.94,A -85,B 0,C 180,E1 20950.303,E2 20950.303} C_VEL
LIN {X 0,Y 489.208,Z 1146.552,A -85,B 0,C 180,E1 20948.036,E2 20948.036} C_VEL
LIN {X 0,Y 492.28,Z 1132.623,A -85,B 0,C 180,E1 20945.905,E2 20945.905} C_VEL
LIN {X 0,Y 495.698,Z 1117.325,A -85,B 0,C 180,E1 20943.914,E2 20943.914} C_VEL
LIN {X 0,Y 499.265,Z 1101.179,A -85,B 0,C 180,E1 20942.12,E2 20942.12} C_VEL
LIN {X 0,Y 502.832,Z 1083.987,A -85,B 0,C 180,E1 20940.519,E2 20940.519} C_VEL
LIN {X 0,Y 506.601,Z 1064.63,A -85,B 0,C 180,E1 20938.994,E2 20938.994} C_VEL
LIN {X 0,Y 509.927,Z 1045.99,A -85,B 0,C 180,E1 20937.769,E2 20937.769} C_VEL
LIN {X 0,Y 512.944,Z 1026.683,A -85,B 0,C 180,E1 20936.728,E2 20936.728} C_VEL
LIN {X 0,Y 515.739,Z 1006.23,A -85,B 0,C 180,E1 20935.824,E2 20935.824} C_VEL
LIN {X 0,Y 517.997,Z 985.502,A -85,B 0,C 180,E1 20935.118,E2 20935.118} C_VEL
LIN {X 0,Y 519.939,Z 962.327,A -85,B 0,C 180,E1 20934.539,E2 20934.539} C_VEL
LIN {X 0,Y 521.055,Z 939.727,A -85,B 0,C 180,E1 20934.155,E2 20934.155} C_VEL
LIN {X 0,Y 527.277,Z 697.87,A -85,B 0,C 180,E1 20930.849,E2 20930.849} C_VEL
LIN {X 0,Y 519.053,Z 644.809,A -85,B 0,C 180,E1 20929.073,E2 20929.073} C_VEL
LIN {X 0,Y 516.268,Z 627.104,A -85,B 0,C 180,E1 20928.409,E2 20928.409} C_VEL
LIN {X 0,Y 520.201,Z 599.816,A -85,B 0,C 180,E1 20926.121,E2 20926.121} C_VEL
LIN {X 0,Y 513.403,Z 581.229,A -85,B 0,C 180,E1 20923.432,E2 20923.432} C_VEL
LIN {X 0,Y 506.123,Z 563.335,A -85,B 0,C 180,E1 20920.54,E2 20920.54} C_VEL
LIN {X 0,Y 499.04,Z 547.593,A -85,B 0,C 180,E1 20917.67,E2 20917.67} C_VEL
LIN {X 0,Y 493.291,Z 535.564,A -85,B 0,C 180,E1 20915.23,E2 20915.23} C_VEL
LIN {X 0,Y 488.633,Z 526.461,A -85,B 0,C 180,E1 20913.185,E2 20913.185} C_VEL
LIN {X 0,Y 486.245,Z 521.909,A -85,B 0,C 180,E1 20912.093,E2 20912.093} C_VEL
LIN {X 0,Y 484.196,Z 517.754,A -85,B 0,C 180,E1 20911.082,E2 20911.082} C_VEL
LIN {X 0,Y 482.286,Z 514.366,A -85,B 0,C 180,E1 20910.174,E2 20910.174} C_VEL
LIN {X 0,Y 482.074,Z 513.283,A -85,B 0,C 180,E1 20909.854,E2 20909.854} C_VEL
LIN {X 0,Y 482.025,Z 513.164,A -85,B 0,C 180,E1 20906.351,E2 20906.351} C_VEL
LIN {X 0,Y 482.023,Z 513.161,A -85,B 0,C 180,E1 20902.695,E2 20902.695} C_VEL
LIN {X 0,Y 482.051,Z 513.156,A -85,B 0,C 180,E1 20899.257,E2 20899.257} C_VEL
LIN {X 0,Y 482.044,Z 513.162,A -85,B 0,C 180,E1 20895.644,E2 20895.644} C_VEL
LIN {X 0,Y 482.018,Z 513.184,A -85,B 0,C 180,E1 20892.094,E2 20892.094} C_VEL
LIN {X 0,Y 482.03,Z 513.186,A -85,B 0,C 180,E1 20888.469,E2 20888.469} C_VEL
LIN {X 0,Y 482.05,Z 513.16,A -85,B 0,C 180,E1 20884.879,E2 20884.879} C_VEL
LIN {X 0,Y 482.033,Z 513.156,A -85,B 0,C 180,E1 20881.307,E2 20881.307} C_VEL
LIN {X 0,Y 482.013,Z 513.175,A -85,B 0,C 180,E1 20877.86,E2 20877.86} C_VEL
LIN {X 0,Y 482.042,Z 513.186,A -85,B 0,C 180,E1 20874.286,E2 20874.286} C_VEL
LIN {X 0,Y 482.05,Z 513.165,A -85,B 0,C 180,E1 20870.689,E2 20870.689} C_VEL
LIN {X 0,Y 482.017,Z 513.159,A -85,B 0,C 180,E1 20867.143,E2 20867.143} C_VEL
LIN {X 0,Y 482.01,Z 513.161,A -85,B 0,C 180,E1 20863.489,E2 20863.489} C_VEL
LIN {X 0,Y 482.047,Z 513.165,A -85,B 0,C 180,E1 20859.985,E2 20859.985} C_VEL
LIN {X 0,Y 482.039,Z 513.174,A -85,B 0,C 180,E1 20856.463,E2 20856.463} C_VEL
LIN {X 0,Y 482.01,Z 513.184,A -85,B 0,C 180,E1 20852.98,E2 20852.98} C_VEL
LIN {X 0,Y 482.061,Z 513.424,A -85,B 0,C 180,E1 20850.445,E2 20850.445} C_VEL
LIN {X 0,Y 483.85,Z 517.335,A -85,B 0,C 180,E1 20849.445,E2 20849.445} C_VEL
LIN {X 0,Y 484.893,Z 519.204,A -85,B 0,C 180,E1 20848.968,E2 20848.968} C_VEL
LIN {X 0,Y 487.516,Z 524.123,A -85,B 0,C 180,E1 20847.774,E2 20847.774} C_VEL
LIN {X 0,Y 490.466,Z 529.861,A -85,B 0,C 180,E1 20846.463,E2 20846.463} C_VEL
LIN {X 0,Y 496.099,Z 540.85,A -85,B 0,C 180,E1 20844.116,E2 20844.116} C_VEL
LIN {X 0,Y 502.611,Z 554.543,A -85,B 0,C 180,E1 20841.542,E2 20841.542} C_VEL
LIN {X 0,Y 516.824,Z 574.84,A -85,B 0,C 180,E1 20839.381,E2 20839.381} C_VEL
LIN {X 0,Y 530.668,Z 596.443,A -85,B 0,C 180,E1 20837.434,E2 20837.434} C_VEL
LIN {X 0,Y 533.842,Z 602.045,A -85,B 0,C 180,E1 20836.998,E2 20836.998} C_VEL
LIN {X 0,Y 524.671,Z 841.664,A -85,B 0,C 180,E1 20833.297,E2 20833.297} C_VEL
LIN {X 0,Y 521.479,Z 924.603,A -85,B 0,C 180,E1 20831.981,E2 20831.981} C_VEL
LIN {X 0,Y 519.697,Z 949.315,A -85,B 0,C 180,E1 20831.411,E2 20831.411} C_VEL
LIN {X 0,Y 517.557,Z 972.651,A -85,B 0,C 180,E1 20830.693,E2 20830.693} C_VEL
LIN {X 0,Y 514.947,Z 995.398,A -85,B 0,C 180,E1 20829.791,E2 20829.791} C_VEL
LIN {X 0,Y 512.091,Z 1017.331,A -85,B 0,C 180,E1 20828.739,E2 20828.739} C_VEL
LIN {X 0,Y 508.767,Z 1039.667,A -85,B 0,C 180,E1 20827.44,E2 20827.44} C_VEL
LIN {X 0,Y 505.593,Z 1059.278,A -85,B 0,C 180,E1 20826.109,E2 20826.109} C_VEL
LIN {X 0,Y 501.944,Z 1080.205,A -85,B 0,C 180,E1 20824.441,E2 20824.441} C_VEL
LIN {X 0,Y 498.579,Z 1098.947,A -85,B 0,C 180,E1 20822.716,E2 20822.716} C_VEL
LIN {X 0,Y 495.123,Z 1117.578,A -85,B 0,C 180,E1 20820.724,E2 20820.724} C_VEL
LIN {X 0,Y 492.085,Z 1133.99,A -85,B 0,C 180,E1 20818.721,E2 20818.721} C_VEL
LIN {X 0,Y 489.177,Z 1150.054,A -85,B 0,C 180,E1 20816.455,E2 20816.455} C_VEL
LIN {X 0,Y 486.774,Z 1163.962,A -85,B 0,C 180,E1 20814.212,E2 20814.212} C_VEL
LIN {X 0,Y 484.606,Z 1177.549,A -85,B 0,C 180,E1 20811.674,E2 20811.674} C_VEL
LIN {X 0,Y 483,Z 1188.672,A -85,B 0,C 180,E1 20809.265,E2 20809.265} C_VEL
LIN {X 0,Y 481.636,Z 1199.878,A -85,B 0,C 180,E1 20806.399,E2 20806.399} C_VEL
LIN {X 0,Y 480.849,Z 1207.837,A -85,B 0,C 180,E1 20803.958,E2 20803.958} C_VEL
LIN {X 0,Y 480.286,Z 1215.582,A -85,B 0,C 180,E1 20801.042,E2 20801.042} C_VEL
LIN {X 0,Y 480.061,Z 1220.545,A -85,B 0,C 180,E1 20798.625,E2 20798.625} C_VEL
LIN {X 0,Y 479.952,Z 1224.643,A -85,B 0,C 180,E1 20795.979,E2 20795.979} C_VEL
LIN {X 0,Y 479.917,Z 1227.247,A -85,B 0,C 180,E1 20793.225,E2 20793.225} C_VEL
LIN {X 0,Y 479.921,Z 1228.227,A -85,B 0,C 180,E1 20790.955,E2 20790.955} C_VEL
LIN {X 0,Y 479.926,Z 1228.13,A -85,B 0,C 180,E1 20788.567,E2 20788.567} C_VEL
LIN {X 0,Y 479.936,Z 1226.412,A -85,B 0,C 180,E1 20785.699,E2 20785.699} C_VEL
LIN {X 0,Y 479.973,Z 1223.63,A -85,B 0,C 180,E1 20783.301,E2 20783.301} C_VEL
LIN {X 0,Y 480.104,Z 1219.235,A -85,B 0,C 180,E1 20780.651,E2 20780.651} C_VEL
LIN {X 0,Y 480.455,Z 1212.882,A -85,B 0,C 180,E1 20777.867,E2 20777.867} C_VEL
LIN {X 0,Y 481.011,Z 1205.975,A -85,B 0,C 180,E1 20775.433,E2 20775.433} C_VEL
LIN {X 0,Y 482.097,Z 1195.811,A -85,B 0,C 180,E1 20772.499,E2 20772.499} C_VEL
LIN {X 0,Y 483.337,Z 1186.182,A -85,B 0,C 180,E1 20770.168,E2 20770.168} C_VEL
LIN {X 0,Y 485.277,Z 1173.177,A -85,B 0,C 180,E1 20767.466,E2 20767.466} C_VEL
LIN {X 0,Y 487.426,Z 1160.05,A -85,B 0,C 180,E1 20765.133,E2 20765.133} C_VEL
LIN {X 0,Y 490.217,Z 1144.19,A -85,B 0,C 180,E1 20762.683,E2 20762.683} C_VEL
LIN {X 0,Y 493.058,Z 1128.679,A -85,B 0,C 180,E1 20760.611,E2 20760.611} C_VEL
LIN {X 0,Y 496.558,Z 1109.726,A -85,B 0,C 180,E1 20758.405,E2 20758.405} C_VEL
LIN {X 0,Y 499.696,Z 1092.632,A -85,B 0,C 180,E1 20756.684,E2 20756.684} C_VEL
LIN {X 0,Y 503.483,Z 1071.459,A -85,B 0,C 180,E1 20754.837,E2 20754.837} C_VEL
LIN {X 0,Y 506.671,Z 1052.535,A -85,B 0,C 180,E1 20753.419,E2 20753.419} C_VEL
LIN {X 0,Y 510.219,Z 1029.771,A -85,B 0,C 180,E1 20751.96,E2 20751.96} C_VEL
LIN {X 0,Y 513.145,Z 1009.153,A -85,B 0,C 180,E1 20750.853,E2 20750.853} C_VEL
LIN {X 0,Y 516.192,Z 984.534,A -85,B 0,C 180,E1 20749.76,E2 20749.76} C_VEL
LIN {X 0,Y 518.467,Z 962.762,A -85,B 0,C 180,E1 20748.987,E2 20748.987} C_VEL
LIN {X 0,Y 520.607,Z 937.486,A -85,B 0,C 180,E1 20748.301,E2 20748.301} C_VEL
LIN {X 0,Y 521.892,Z 915.509,A -85,B 0,C 180,E1 20747.866,E2 20747.866} C_VEL
LIN {X 0,Y 531.081,Z 671.392,A -85,B 0,C 180,E1 20744.066,E2 20744.066} C_VEL
LIN {X 0,Y 533.674,Z 601.395,A -85,B 0,C 180,E1 20742.981,E2 20742.981} C_VEL
LIN {X 0,Y 520.192,Z 579.927,A -85,B 0,C 180,E1 20741.119,E2 20741.119} C_VEL
LIN {X 0,Y 507.419,Z 561.327,A -85,B 0,C 180,E1 20739.238,E2 20739.238} C_VEL
LIN {X 0,Y 502.291,Z 553.972,A -85,B 0,C 180,E1 20738.396,E2 20738.396} C_VEL
LIN {X 0,Y 495.789,Z 540.277,A -85,B 0,C 180,E1 20735.793,E2 20735.793} C_VEL
LIN {X 0,Y 490.67,Z 530.269,A -85,B 0,C 180,E1 20733.662,E2 20733.662} C_VEL
LIN {X 0,Y 488.76,Z 526.574,A -85,B 0,C 180,E1 20732.829,E2 20732.829} C_VEL
LIN {X 0,Y 486.375,Z 521.994,A -85,B 0,C 180,E1 20731.755,E2 20731.755} C_VEL
LIN {X 0,Y 484.06,Z 517.604,A -85,B 0,C 180,E1 20730.678,E2 20730.678} C_VEL
LIN {X 0,Y 482.154,Z 513.844,A -85,B 0,C 180,E1 20729.712,E2 20729.712} C_VEL
LIN {X 0,Y 482.029,Z 513.248,A -85,B 0,C 180,E1 20729.403,E2 20729.403} C_VEL
LIN {X 0,Y 482.054,Z 513.17,A -85,B 0,C 180,E1 20725.955,E2 20725.955} C_VEL
LIN {X 0,Y 482.023,Z 513.18,A -85,B 0,C 180,E1 20722.438,E2 20722.438} C_VEL
LIN {X 0,Y 482.015,Z 513.19,A -85,B 0,C 180,E1 20718.881,E2 20718.881} C_VEL
LIN {X 0,Y 482.045,Z 513.179,A -85,B 0,C 180,E1 20715.274,E2 20715.274} C_VEL
LIN {X 0,Y 482.047,Z 513.16,A -85,B 0,C 180,E1 20711.729,E2 20711.729} C_VEL
LIN {X 0,Y 482.013,Z 513.155,A -85,B 0,C 180,E1 20708.229,E2 20708.229} C_VEL
LIN {X 0,Y 482.023,Z 513.166,A -85,B 0,C 180,E1 20704.64,E2 20704.64} C_VEL
LIN {X 0,Y 482.058,Z 513.185,A -85,B 0,C 180,E1 20701.07,E2 20701.07} C_VEL
LIN {X 0,Y 482.039,Z 513.171,A -85,B 0,C 180,E1 20697.503,E2 20697.503} C_VEL
LIN {X 0,Y 482.017,Z 513.158,A -85,B 0,C 180,E1 20693.927,E2 20693.927} C_VEL
LIN {X 0,Y 482.038,Z 513.16,A -85,B 0,C 180,E1 20690.448,E2 20690.448} C_VEL
LIN {X 0,Y 482.054,Z 513.177,A -85,B 0,C 180,E1 20686.811,E2 20686.811} C_VEL
LIN {X 0,Y 482.039,Z 513.186,A -85,B 0,C 180,E1 20683.242,E2 20683.242} C_VEL
LIN {X 0,Y 482.024,Z 513.176,A -85,B 0,C 180,E1 20679.605,E2 20679.605} C_VEL
LIN {X 0,Y 482.048,Z 513.164,A -85,B 0,C 180,E1 20676.141,E2 20676.141} C_VEL
LIN {X 0,Y 482.054,Z 513.164,A -85,B 0,C 180,E1 20672.582,E2 20672.582} C_VEL
LIN {X 0,Y 482.093,Z 513.422,A -85,B 0,C 180,E1 20669.917,E2 20669.917} C_VEL
LIN {X 0,Y 483.594,Z 517.014,A -85,B 0,C 180,E1 20669.013,E2 20669.013} C_VEL
LIN {X 0,Y 484.718,Z 518.692,A -85,B 0,C 180,E1 20668.54,E2 20668.54} C_VEL
LIN {X 0,Y 486.768,Z 522.581,A -85,B 0,C 180,E1 20667.579,E2 20667.579} C_VEL
LIN {X 0,Y 490.096,Z 529.436,A -85,B 0,C 180,E1 20666.012,E2 20666.012} C_VEL
LIN {X 0,Y 493.988,Z 536.995,A -85,B 0,C 180,E1 20664.342,E2 20664.342} C_VEL
LIN {X 0,Y 500.235,Z 550.232,A -85,B 0,C 180,E1 20661.71,E2 20661.71} C_VEL
LIN {X 0,Y 506.753,Z 564.979,A -85,B 0,C 180,E1 20659.074,E2 20659.074} C_VEL
LIN {X 0,Y 513.782,Z 582.29,A -85,B 0,C 180,E1 20656.3,E2 20656.3} C_VEL
LIN {X 0,Y 520.137,Z 599.704,A -85,B 0,C 180,E1 20653.791,E2 20653.791} C_VEL
LIN {X 0,Y 516.224,Z 628.101,A -85,B 0,C 180,E1 20651.434,E2 20651.434} C_VEL
LIN {X 0,Y 525.109,Z 683.694,A -85,B 0,C 180,E1 20649.504,E2 20649.504} C_VEL
LIN {X 0,Y 527.265,Z 699.498,A -85,B 0,C 180,E1 20649.021,E2 20649.021} C_VEL
LIN {X 0,Y 520.537,Z 951.818,A -85,B 0,C 180,E1 20645.562,E2 20645.562} C_VEL
LIN {X 0,Y 518.985,Z 974.059,A -85,B 0,C 180,E1 20645.098,E2 20645.098} C_VEL
LIN {X 0,Y 516.971,Z 995.09,A -85,B 0,C 180,E1 20644.485,E2 20644.485} C_VEL
LIN {X 0,Y 514.48,Z 1015.329,A -85,B 0,C 180,E1 20643.7,E2 20643.7} C_VEL
LIN {X 0,Y 511.378,Z 1036.69,A -85,B 0,C 180,E1 20642.659,E2 20642.659} C_VEL
LIN {X 0,Y 508.144,Z 1056.188,A -85,B 0,C 180,E1 20641.494,E2 20641.494} C_VEL
LIN {X 0,Y 504.637,Z 1074.694,A -85,B 0,C 180,E1 20640.15,E2 20640.15} C_VEL
LIN {X 0,Y 500.92,Z 1093.125,A -85,B 0,C 180,E1 20638.563,E2 20638.563} C_VEL
LIN {X 0,Y 498.928,Z 1102.519,A -85,B 0,C 180,E1 20637.641,E2 20637.641} C_VEL
LIN {X 0,Y 496.774,Z 1108.315,A -85,B 0,C 180,E1 20637.082,E2 20637.082} C_VEL
LIN {X 0,Y 488.207,Z 1122.516,A -85,B 0,C 180,E1 20635.754,E2 20635.754} C_VEL
LIN {X 0,Y 486.127,Z 1127.636,A -85,B 0,C 180,E1 20635.13,E2 20635.13} C_VEL
LIN {X 0,Y 482.812,Z 1141.833,A -85,B 0,C 180,E1 20633.042,E2 20633.042} C_VEL
LIN {X 0,Y 479.958,Z 1154.454,A -85,B 0,C 180,E1 20630.869,E2 20630.869} C_VEL
LIN {X 0,Y 477.49,Z 1165.663,A -85,B 0,C 180,E1 20628.559,E2 20628.559} C_VEL
LIN {X 0,Y 475.409,Z 1176.128,A -85,B 0,C 180,E1 20625.993,E2 20625.993} C_VEL
LIN {X 0,Y 473.929,Z 1184.715,A -85,B 0,C 180,E1 20623.419,E2 20623.419} C_VEL
LIN {X 0,Y 472.956,Z 1191.511,A -85,B 0,C 180,E1 20620.845,E2 20620.845} C_VEL
LIN {X 0,Y 472.358,Z 1197.042,A -85,B 0,C 180,E1 20618.153,E2 20618.153} C_VEL
LIN {X 0,Y 472.087,Z 1200.728,A -85,B 0,C 180,E1 20615.591,E2 20615.591} C_VEL
LIN {X 0,Y 471.977,Z 1203.194,A -85,B 0,C 180,E1 20612.793,E2 20612.793} C_VEL
LIN {X 0,Y 471.956,Z 1204.063,A -85,B 0,C 180,E1 20610.121,E2 20610.121} C_VEL
LIN {X 0,Y 471.97,Z 1203.372,A -85,B 0,C 180,E1 20607.45,E2 20607.45} C_VEL
LIN {X 0,Y 472.058,Z 1201.299,A -85,B 0,C 180,E1 20604.774,E2 20604.774} C_VEL
LIN {X 0,Y 472.311,Z 1197.585,A -85,B 0,C 180,E1 20602.091,E2 20602.091} C_VEL
LIN {X 0,Y 472.893,Z 1192.025,A -85,B 0,C 180,E1 20599.277,E2 20599.277} C_VEL
LIN {X 0,Y 473.89,Z 1185.018,A -85,B 0,C 180,E1 20596.58,E2 20596.58} C_VEL
LIN {X 0,Y 475.351,Z 1176.465,A -85,B 0,C 180,E1 20594.005,E2 20594.005} C_VEL
LIN {X 0,Y 477.414,Z 1166.084,A -85,B 0,C 180,E1 20591.438,E2 20591.438} C_VEL
LIN {X 0,Y 479.862,Z 1154.948,A -85,B 0,C 180,E1 20589.127,E2 20589.127} C_VEL
LIN {X 0,Y 482.858,Z 1141.724,A -85,B 0,C 180,E1 20586.843,E2 20586.843} C_VEL
LIN {X 0,Y 486.302,Z 1126.955,A -85,B 0,C 180,E1 20584.681,E2 20584.681} C_VEL
LIN {X 0,Y 489.968,Z 1111.297,A -85,B 0,C 180,E1 20582.734,E2 20582.734} C_VEL
LIN {X 0,Y 493.697,Z 1094.519,A -85,B 0,C 180,E1 20580.985,E2 20580.985} C_VEL
LIN {X 0,Y 497.758,Z 1075.265,A -85,B 0,C 180,E1 20579.29,E2 20579.29} C_VEL
LIN {X 0,Y 501.469,Z 1056.412,A -85,B 0,C 180,E1 20577.903,E2 20577.903} C_VEL
LIN {X 0,Y 504.815,Z 1036.944,A -85,B 0,C 180,E1 20576.727,E2 20576.727} C_VEL
LIN {X 0,Y 508.093,Z 1015.237,A -85,B 0,C 180,E1 20575.658,E2 20575.658} C_VEL
LIN {X 0,Y 510.76,Z 994.326,A -85,B 0,C 180,E1 20574.843,E2 20574.843} C_VEL
LIN {X 0,Y 512.856,Z 972.915,A -85,B 0,C 180,E1 20574.223,E2 20574.223} C_VEL
LIN {X 0,Y 514.463,Z 949.576,A -85,B 0,C 180,E1 20573.747,E2 20573.747} C_VEL
LIN {X 0,Y 521.364,Z 699.357,A -85,B 0,C 180,E1 20570.275,E2 20570.275} C_VEL
LIN {X 0,Y 513.399,Z 647.012,A -85,B 0,C 180,E1 20568.491,E2 20568.491} C_VEL
LIN {X 0,Y 510.142,Z 626.426,A -85,B 0,C 180,E1 20567.716,E2 20567.716} C_VEL
LIN {X 0,Y 513.574,Z 603.37,A -85,B 0,C 180,E1 20565.764,E2 20565.764} C_VEL
LIN {X 0,Y 506.872,Z 584.915,A -85,B 0,C 180,E1 20563.043,E2 20563.043} C_VEL
LIN {X 0,Y 499.974,Z 567.9,A -85,B 0,C 180,E1 20560.238,E2 20560.238} C_VEL
LIN {X 0,Y 493.284,Z 552.841,A -85,B 0,C 180,E1 20557.453,E2 20557.453} C_VEL
LIN {X 0,Y 487.718,Z 541.074,A -85,B 0,C 180,E1 20555.033,E2 20555.033} C_VEL
LIN {X 0,Y 483.14,Z 532.053,A -85,B 0,C 180,E1 20552.977,E2 20552.977} C_VEL
LIN {X 0,Y 480.81,Z 527.567,A -85,B 0,C 180,E1 20551.885,E2 20551.885} C_VEL
LIN {X 0,Y 478.785,Z 523.5,A -85,B 0,C 180,E1 20550.874,E2 20550.874} C_VEL
LIN {X 0,Y 476.906,Z 519.936,A -85,B 0,C 180,E1 20549.934,E2 20549.934} C_VEL
LIN {X 0,Y 475.601,Z 517.9,A -85,B 0,C 180,E1 20549.331,E2 20549.331} C_VEL
LIN {X 0,Y 474.109,Z 514.312,A -85,B 0,C 180,E1 20548.328,E2 20548.328} C_VEL
LIN {X 0,Y 474.086,Z 514.176,A -85,B 0,C 180,E1 20544.683,E2 20544.683} C_VEL
LIN {X 0,Y 474.115,Z 514.174,A -85,B 0,C 180,E1 20541.139,E2 20541.139} C_VEL
LIN {X 0,Y 474.116,Z 514.164,A -85,B 0,C 180,E1 20537.426,E2 20537.426} C_VEL
LIN {X 0,Y 474.09,Z 514.153,A -85,B 0,C 180,E1 20533.788,E2 20533.788} C_VEL
LIN {X 0,Y 474.077,Z 514.145,A -85,B 0,C 180,E1 20530.205,E2 20530.205} C_VEL
LIN {X 0,Y 474.103,Z 514.149,A -85,B 0,C 180,E1 20526.63,E2 20526.63} C_VEL
LIN {X 0,Y 474.112,Z 514.169,A -85,B 0,C 180,E1 20523.022,E2 20523.022} C_VEL
LIN {X 0,Y 474.088,Z 514.17,A -85,B 0,C 180,E1 20519.396,E2 20519.396} C_VEL
LIN {X 0,Y 474.071,Z 514.15,A -85,B 0,C 180,E1 20515.767,E2 20515.767} C_VEL
LIN {X 0,Y 474.102,Z 514.142,A -85,B 0,C 180,E1 20512.243,E2 20512.243} C_VEL
LIN {X 0,Y 474.107,Z 514.158,A -85,B 0,C 180,E1 20508.689,E2 20508.689} C_VEL
LIN {X 0,Y 474.073,Z 514.179,A -85,B 0,C 180,E1 20505.214,E2 20505.214} C_VEL
LIN {X 0,Y 474.079,Z 514.168,A -85,B 0,C 180,E1 20501.556,E2 20501.556} C_VEL
LIN {X 0,Y 474.117,Z 514.154,A -85,B 0,C 180,E1 20497.951,E2 20497.951} C_VEL
LIN {X 0,Y 474.098,Z 514.154,A -85,B 0,C 180,E1 20494.383,E2 20494.383} C_VEL
